LIN {X 0,Y 342.196,Z 1212.787,A -85,B 0,C 180,E1 21187.644,E2 21187.644} C_VEL
LIN {X 0,Y 370.541,Z 1183.05,A -85,B 0,C 180,E1 21194.239,E2 21194.239} C_VEL
LIN {X 0,Y 337.075,Z 1218.846,A -85,B 0,C 180,E1 21204.188,E2 21204.188} C_VEL
LIN {X 0,Y 317.104,Z 1240.275,A -85,B 0,C 180,E1 21216.022,E2 21216.022} C_VEL
LIN {X 0,Y 309.368,Z 1248.117,A -85,B 0,C 180,E1 21227.294,E2 21227.294} C_VEL
LIN {X 0,Y 299.7,Z 1248.319,A -85,B 0,C 180,E1 21233.729,E2 21233.729} C_VEL
LIN {X 0,Y 299.965,Z 1240.133,A -85,B 0,C 180,E1 21244.381,E2 21244.381} C_VEL
LIN {X 0,Y 304.172,Z 1219.099,A -85,B 0,C 180,E1 21255.958,E2 21255.958} C_VEL
LIN {X 0,Y 314.8,Z 1183.171,A -85,B 0,C 180,E1 21267.012,E2 21267.012} C_VEL
LIN {X 0,Y 330.638,Z 1134.667,A -85,B 0,C 180,E1 21275.905,E2 21275.905} C_VEL
LIN {X 0,Y 345.711,Z 1077.076,A -85,B 0,C 180,E1 21282.387,E2 21282.387} C_VEL
LIN {X 0,Y 328.382,Z 1020.895,A -85,B 0,C 180,E1 21289.392,E2 21289.392} C_VEL
LIN {X 0,Y 317.3,Z 992.068,A -85,B 0,C 180,E1 21293.134,E2 21293.134} C_VEL
LIN {X 0,Y 333.633,Z 1036.761,A -85,B 0,C 180,E1 21296.365,E2 21296.365} C_VEL
LIN {X 0,Y 329.633,Z 1087.019,A -85,B 0,C 180,E1 21298.729,E2 21298.729} C_VEL
LIN {X 0,Y 321.057,Z 1131.238,A -85,B 0,C 180,E1 21303.54,E2 21303.54} C_VEL
LIN {X 0,Y 311.784,Z 1164.217,A -85,B 0,C 180,E1 21310.381,E2 21310.381} C_VEL
LIN {X 0,Y 304.757,Z 1185.316,A -85,B 0,C 180,E1 21319.168,E2 21319.168} C_VEL
LIN {X 0,Y 302.413,Z 1192.13,A -85,B 0,C 180,E1 21328.492,E2 21328.492} C_VEL
LIN {X 0,Y 304.538,Z 1184.356,A -85,B 0,C 180,E1 21338.525,E2 21338.525} C_VEL
LIN {X 0,Y 311.172,Z 1162.189,A -85,B 0,C 180,E1 21347.305,E2 21347.305} C_VEL
LIN {X 0,Y 320.195,Z 1127.219,A -85,B 0,C 180,E1 21354.236,E2 21354.236} C_VEL
LIN {X 0,Y 327.949,Z 1082.319,A -85,B 0,C 180,E1 21358.849,E2 21358.849} C_VEL
LIN {X 0,Y 330.843,Z 1031.167,A -85,B 0,C 180,E1 21361.083,E2 21361.083} C_VEL
LIN {X 0,Y 306.991,Z 970.809,A -85,B 0,C 180,E1 21365.672,E2 21365.672} C_VEL
LIN {X 0,Y 296.216,Z 948.94,A -85,B 0,C 180,E1 21368,E2 21368} C_VEL
LIN {X 0,Y 296.219,Z 948.94,A -85,B 0,C 180,E1 21380.134,E2 21380.134} C_VEL
LIN {X 0,Y 296.775,Z 948.94,A -85,B 0,C 180,E1 21393.307,E2 21393.307} C_VEL
LIN {X 0,Y 298.047,Z 948.94,A -85,B 0,C 180,E1 21406.723,E2 21406.723} C_VEL
LIN {X 0,Y 298.821,Z 948.94,A -85,B 0,C 180,E1 21418.516,E2 21418.516} C_VEL
LIN {X 0,Y 297.907,Z 948.94,A -85,B 0,C 180,E1 21430.243,E2 21430.243} C_VEL
LIN {X 0,Y 297.236,Z 950.399,A -85,B 0,C 180,E1 21441.304,E2 21441.304} C_VEL
LIN {X 0,Y 327.096,Z 1016.083,A -85,B 0,C 180,E1 21452.614,E2 21452.614} C_VEL
LIN {X 0,Y 351.234,Z 1081.655,A -85,B 0,C 180,E1 21462.15,E2 21462.15} C_VEL
LIN {X 0,Y 328.608,Z 1154.976,A -85,B 0,C 180,E1 21469.978,E2 21469.978} C_VEL
LIN {X 0,Y 311.576,Z 1211.957,A -85,B 0,C 180,E1 21479.926,E2 21479.926} C_VEL
LIN {X 0,Y 302.573,Z 1251.413,A -85,B 0,C 180,E1 21491.052,E2 21491.052} C_VEL
LIN {X 0,Y 300.193,Z 1272.803,A -85,B 0,C 180,E1 21501.423,E2 21501.423} C_VEL
LIN {X 0,Y 299.986,Z 1281.152,A -85,B 0,C 180,E1 21511.521,E2 21511.521} C_VEL
LIN {X 0,Y 300.221,Z 1277.634,A -85,B 0,C 180,E1 21521.736,E2 21521.736} C_VEL
LIN {X 0,Y 307.735,Z 1258.286,A -85,B 0,C 180,E1 21534.221,E2 21534.221} C_VEL
LIN {X 0,Y 339.314,Z 1212.711,A -85,B 0,C 180,E1 21549.251,E2 21549.251} C_VEL
LIN {X 0,Y 361.602,Z 1191.419,A -85,B 0,C 180,E1 21554.373,E2 21554.373} C_VEL
LIN {X 0,Y 327.946,Z 1224.179,A -85,B 0,C 180,E1 21564.685,E2 21564.685} C_VEL
LIN {X 0,Y 307.047,Z 1244.419,A -85,B 0,C 180,E1 21578.268,E2 21578.268} C_VEL
LIN {X 0,Y 300.37,Z 1249.085,A -85,B 0,C 180,E1 21590.489,E2 21590.489} C_VEL
LIN {X 0,Y 299.7,Z 1248.319,A -85,B 0,C 180,E1 21593.729,E2 21593.729} C_VEL
LIN {X 0,Y 291.795,Z 1244.564,A -85,B 0,C 180,E1 21600.397,E2 21600.397} C_VEL
LIN {X 0,Y 294.315,Z 1227.603,A -85,B 0,C 180,E1 21612.345,E2 21612.345} C_VEL
LIN {X 0,Y 303.211,Z 1196.172,A -85,B 0,C 180,E1 21624.03,E2 21624.03} C_VEL
LIN {X 0,Y 317.833,Z 1152.021,A -85,B 0,C 180,E1 21633.753,E2 21633.753} C_VEL
LIN {X 0,Y 334.741,Z 1096.51,A -85,B 0,C 180,E1 21641.141,E2 21641.141} C_VEL
LIN {X 0,Y 337.819,Z 1076.712,A -85,B 0,C 180,E1 21643.202,E2 21643.202} C_VEL
LIN {X 0,Y 320.249,Z 1020.145,A -85,B 0,C 180,E1 21650.453,E2 21650.453} C_VEL
LIN {X 0,Y 313.932,Z 1002.402,A -85,B 0,C 180,E1 21652.96,E2 21652.96} C_VEL
LIN {X 0,Y 326.976,Z 1038.863,A -85,B 0,C 180,E1 21655.637,E2 21655.637} C_VEL
LIN {X 0,Y 322.812,Z 1088.072,A -85,B 0,C 180,E1 21658.019,E2 21658.019} C_VEL
LIN {X 0,Y 313.933,Z 1132.251,A -85,B 0,C 180,E1 21662.919,E2 21662.919} C_VEL
LIN {X 0,Y 303.873,Z 1166.286,A -85,B 0,C 180,E1 21670.229,E2 21670.229} C_VEL
LIN {X 0,Y 296.971,Z 1186.242,A -85,B 0,C 180,E1 21678.881,E2 21678.881} C_VEL
LIN {X 0,Y 294.475,Z 1193.081,A -85,B 0,C 180,E1 21688.451,E2 21688.451} C_VEL
LIN {X 0,Y 296.71,Z 1185.329,A -85,B 0,C 180,E1 21698.751,E2 21698.751} C_VEL
LIN {X 0,Y 303.512,Z 1163.552,A -85,B 0,C 180,E1 21707.65,E2 21707.65} C_VEL
LIN {X 0,Y 312.647,Z 1129.383,A -85,B 0,C 180,E1 21714.669,E2 21714.669} C_VEL
LIN {X 0,Y 320.8,Z 1085.261,A -85,B 0,C 180,E1 21719.404,E2 21719.404} C_VEL
LIN {X 0,Y 324.209,Z 1033.506,A -85,B 0,C 180,E1 21721.77,E2 21721.77} C_VEL
LIN {X 0,Y 300.618,Z 973.534,A -85,B 0,C 180,E1 21726.512,E2 21726.512} C_VEL
LIN {X 0,Y 288.132,Z 948.94,A -85,B 0,C 180,E1 21729.426,E2 21729.426} C_VEL
LIN {X 0,Y 288.256,Z 948.94,A -85,B 0,C 180,E1 21742.696,E2 21742.696} C_VEL
LIN {X 0,Y 288.788,Z 948.94,A -85,B 0,C 180,E1 21753.432,E2 21753.432} C_VEL
LIN {X 0,Y 289.956,Z 948.94,A -85,B 0,C 180,E1 21766.345,E2 21766.345} C_VEL
LIN {X 0,Y 290.838,Z 948.94,A -85,B 0,C 180,E1 21778.475,E2 21778.475} C_VEL
LIN {X 0,Y 289.84,Z 948.94,A -85,B 0,C 180,E1 21790.531,E2 21790.531} C_VEL
LIN {X 0,Y 289.433,Z 950.977,A -85,B 0,C 180,E1 21799.772,E2 21799.772} C_VEL
LIN {X 0,Y 318.268,Z 1014.18,A -85,B 0,C 180,E1 21811.209,E2 21811.209} C_VEL
LIN {X 0,Y 343.351,Z 1082.536,A -85,B 0,C 180,E1 21821.496,E2 21821.496} C_VEL
LIN {X 0,Y 320.993,Z 1155.423,A -85,B 0,C 180,E1 21829.546,E2 21829.546} C_VEL
LIN {X 0,Y 303.671,Z 1211.944,A -85,B 0,C 180,E1 21839.692,E2 21839.692} C_VEL
LIN {X 0,Y 294.557,Z 1251.213,A -85,B 0,C 180,E1 21851.101,E2 21851.101} C_VEL
LIN {X 0,Y 292.141,Z 1273.544,A -85,B 0,C 180,E1 21862.614,E2 21862.614} C_VEL
LIN {X 0,Y 292.001,Z 1280.42,A -85,B 0,C 180,E1 21871.562,E2 21871.562} C_VEL
LIN {X 0,Y 292.314,Z 1277.354,A -85,B 0,C 180,E1 21882.058,E2 21882.058} C_VEL
LIN {X 0,Y 301.034,Z 1257.777,A -85,B 0,C 180,E1 21895.446,E2 21895.446} C_VEL
LIN {X 0,Y 337.978,Z 1211.874,A -85,B 0,C 180,E1 21911.122,E2 21911.122} C_VEL
LIN {X 0,Y 352.937,Z 1198.914,A -85,B 0,C 180,E1 21914.182,E2 21914.182} C_VEL
LIN {X 0,Y 316.008,Z 1231.474,A -85,B 0,C 180,E1 21926.504,E2 21926.504} C_VEL
LIN {X 0,Y 297.02,Z 1247.559,A -85,B 0,C 180,E1 21940.631,E2 21940.631} C_VEL
LIN {X 0,Y 291.722,Z 1248.78,A -85,B 0,C 180,E1 21953.691,E2 21953.691} C_VEL
LIN {X 0,Y 291.795,Z 1244.564,A -85,B 0,C 180,E1 21960.397,E2 21960.397} C_VEL
LIN {X 0,Y 284.739,Z 1236.825,A -85,B 0,C 180,E1 21967.153,E2 21967.153} C_VEL
LIN {X 0,Y 290.083,Z 1212.471,A -85,B 0,C 180,E1 21979.119,E2 21979.119} C_VEL
LIN {X 0,Y 302.781,Z 1173.653,A -85,B 0,C 180,E1 21990.118,E2 21990.118} C_VEL
LIN {X 0,Y 320.044,Z 1122.033,A -85,B 0,C 180,E1 21998.853,E2 21998.853} C_VEL
LIN {X 0,Y 330.785,Z 1079.888,A -85,B 0,C 180,E1 22003.558,E2 22003.558} C_VEL
LIN {X 0,Y 313.837,Z 1023.996,A -85,B 0,C 180,E1 22010.973,E2 22010.973} C_VEL
LIN {X 0,Y 310.27,Z 1012.617,A -85,B 0,C 180,E1 22012.738,E2 22012.738} C_VEL
LIN {X 0,Y 320.333,Z 1041.652,A -85,B 0,C 180,E1 22014.893,E2 22014.893} C_VEL
LIN {X 0,Y 315.625,Z 1091.457,A -85,B 0,C 180,E1 22017.46,E2 22017.46} C_VEL
LIN {X 0,Y 306.576,Z 1134.252,A -85,B 0,C 180,E1 22022.42,E2 22022.42} C_VEL
LIN {X 0,Y 296.413,Z 1167.185,A -85,B 0,C 180,E1 22029.71,E2 22029.71} C_VEL
LIN {X 0,Y 289.181,Z 1187.17,A -85,B 0,C 180,E1 22038.577,E2 22038.577} C_VEL
LIN {X 0,Y 286.556,Z 1194.03,A -85,B 0,C 180,E1 22048.408,E2 22048.408} C_VEL
LIN {X 0,Y 288.861,Z 1186.306,A -85,B 0,C 180,E1 22058.991,E2 22058.991} C_VEL
LIN {X 0,Y 296.181,Z 1163.803,A -85,B 0,C 180,E1 22068.329,E2 22068.329} C_VEL
LIN {X 0,Y 305.803,Z 1129.297,A -85,B 0,C 180,E1 22075.456,E2 22075.456} C_VEL
LIN {X 0,Y 314.225,Z 1084.222,A -85,B 0,C 180,E1 22080.267,E2 22080.267} C_VEL
LIN {X 0,Y 316.797,Z 1033.119,A -85,B 0,C 180,E1 22082.658,E2 22082.658} C_VEL
LIN {X 0,Y 293.924,Z 975.892,A -85,B 0,C 180,E1 22087.46,E2 22087.46} C_VEL
LIN {X 0,Y 280.112,Z 948.94,A -85,B 0,C 180,E1 22090.95,E2 22090.95} C_VEL
LIN {X 0,Y 280.293,Z 948.94,A -85,B 0,C 180,E1 22105.312,E2 22105.312} C_VEL
LIN {X 0,Y 280.899,Z 948.94,A -85,B 0,C 180,E1 22116.06,E2 22116.06} C_VEL
LIN {X 0,Y 282.11,Z 948.94,A -85,B 0,C 180,E1 22129.115,E2 22129.115} C_VEL
LIN {X 0,Y 282.659,Z 948.94,A -85,B 0,C 180,E1 22141.508,E2 22141.508} C_VEL
LIN {X 0,Y 281.508,Z 948.94,A -85,B 0,C 180,E1 22154.01,E2 22154.01} C_VEL
LIN {X 0,Y 281.347,Z 950.523,A -85,B 0,C 180,E1 22157.992,E2 22157.992} C_VEL
LIN {X 0,Y 310.074,Z 1013.728,A -85,B 0,C 180,E1 22169.983,E2 22169.983} C_VEL
LIN {X 0,Y 334.573,Z 1080.888,A -85,B 0,C 180,E1 22180.455,E2 22180.455} C_VEL
LIN {X 0,Y 334.131,Z 1092.54,A -85,B 0,C 180,E1 22181.816,E2 22181.816} C_VEL
LIN {X 0,Y 310.895,Z 1163.485,A -85,B 0,C 180,E1 22190.258,E2 22190.258} C_VEL
LIN {X 0,Y 293.881,Z 1218.737,A -85,B 0,C 180,E1 22201.116,E2 22201.116} C_VEL
LIN {X 0,Y 285.978,Z 1255.72,A -85,B 0,C 180,E1 22213.112,E2 22213.112} C_VEL
LIN {X 0,Y 284.109,Z 1274.249,A -85,B 0,C 180,E1 22223.945,E2 22223.945} C_VEL
LIN {X 0,Y 283.672,Z 1280.07,A -85,B 0,C 180,E1 22234.678,E2 22234.678} C_VEL
LIN {X 0,Y 285.91,Z 1272.693,A -85,B 0,C 180,E1 22247.049,E2 22247.049} C_VEL
LIN {X 0,Y 302.716,Z 1245.944,A -85,B 0,C 180,E1 22261.838,E2 22261.838} C_VEL
LIN {X 0,Y 343.886,Z 1206.254,A -85,B 0,C 180,E1 22274.536,E2 22274.536} C_VEL
LIN {X 0,Y 307.499,Z 1235.138,A -85,B 0,C 180,E1 22286.657,E2 22286.657} C_VEL
LIN {X 0,Y 289.451,Z 1248.6,A -85,B 0,C 180,E1 22300.103,E2 22300.103} C_VEL
LIN {X 0,Y 283.988,Z 1249.777,A -85,B 0,C 180,E1 22312.352,E2 22312.352} C_VEL
LIN {X 0,Y 284.028,Z 1240.244,A -85,B 0,C 180,E1 22324.628,E2 22324.628} C_VEL
LIN {X 0,Y 284.739,Z 1236.825,A -85,B 0,C 180,E1 22327.153,E2 22327.153} C_VEL
LIN {X 0,Y 279.071,Z 1225.354,A -85,B 0,C 180,E1 22333.898,E2 22333.898} C_VEL
LIN {X 0,Y 289.115,Z 1191.74,A -85,B 0,C 180,E1 22346.116,E2 22346.116} C_VEL
LIN {X 0,Y 305.633,Z 1144.511,A -85,B 0,C 180,E1 22356.172,E2 22356.172} C_VEL
LIN {X 0,Y 323.653,Z 1086.172,A -85,B 0,C 180,E1 22363.538,E2 22363.538} C_VEL
LIN {X 0,Y 310.199,Z 1035.79,A -85,B 0,C 180,E1 22370.437,E2 22370.437} C_VEL
LIN {X 0,Y 306.497,Z 1022.683,A -85,B 0,C 180,E1 22372.489,E2 22372.489} C_VEL
LIN {X 0,Y 313.752,Z 1044.285,A -85,B 0,C 180,E1 22374.122,E2 22374.122} C_VEL
LIN {X 0,Y 308.721,Z 1093.794,A -85,B 0,C 180,E1 22376.8,E2 22376.8} C_VEL
LIN {X 0,Y 299.044,Z 1136.855,A -85,B 0,C 180,E1 22382.011,E2 22382.011} C_VEL
LIN {X 0,Y 288.492,Z 1169.258,A -85,B 0,C 180,E1 22389.529,E2 22389.529} C_VEL
LIN {X 0,Y 280.922,Z 1189.149,A -85,B 0,C 180,E1 22399.026,E2 22399.026} C_VEL
LIN {X 0,Y 278.645,Z 1194.978,A -85,B 0,C 180,E1 22408.363,E2 22408.363} C_VEL
LIN {X 0,Y 281.038,Z 1187.279,A -85,B 0,C 180,E1 22419.244,E2 22419.244} C_VEL
LIN {X 0,Y 288.65,Z 1164.809,A -85,B 0,C 180,E1 22428.825,E2 22428.825} C_VEL
LIN {X 0,Y 298.653,Z 1130.336,A -85,B 0,C 180,E1 22436.11,E2 22436.11} C_VEL
LIN {X 0,Y 307.275,Z 1086.268,A -85,B 0,C 180,E1 22440.945,E2 22440.945} C_VEL
LIN {X 0,Y 310.328,Z 1035.651,A -85,B 0,C 180,E1 22443.398,E2 22443.398} C_VEL
LIN {X 0,Y 287.811,Z 979.04,A -85,B 0,C 180,E1 22448.345,E2 22448.345} C_VEL
LIN {X 0,Y 271.994,Z 948.94,A -85,B 0,C 180,E1 22452.697,E2 22452.697} C_VEL
LIN {X 0,Y 272.115,Z 948.94,A -85,B 0,C 180,E1 22464.111,E2 22464.111} C_VEL
LIN {X 0,Y 272.911,Z 948.94,A -85,B 0,C 180,E1 22476.342,E2 22476.342} C_VEL
LIN {X 0,Y 274.047,Z 948.94,A -85,B 0,C 180,E1 22488.791,E2 22488.791} C_VEL
LIN {X 0,Y 274.647,Z 948.94,A -85,B 0,C 180,E1 22501.552,E2 22501.552} C_VEL
LIN {X 0,Y 273.423,Z 948.94,A -85,B 0,C 180,E1 22514.434,E2 22514.434} C_VEL
LIN {X 0,Y 273.525,Z 951.065,A -85,B 0,C 180,E1 22516.283,E2 22516.283} C_VEL
LIN {X 0,Y 299.882,Z 1008.76,A -85,B 0,C 180,E1 22527.884,E2 22527.884} C_VEL
LIN {X 0,Y 323.347,Z 1071.686,A -85,B 0,C 180,E1 22538.212,E2 22538.212} C_VEL
LIN {X 0,Y 327.574,Z 1091.222,A -85,B 0,C 180,E1 22541.025,E2 22541.025} C_VEL
LIN {X 0,Y 303.72,Z 1162.326,A -85,B 0,C 180,E1 22549.594,E2 22549.594} C_VEL
LIN {X 0,Y 286.233,Z 1217.541,A -85,B 0,C 180,E1 22560.633,E2 22560.633} C_VEL
LIN {X 0,Y 278.212,Z 1254.069,A -85,B 0,C 180,E1 22572.626,E2 22572.626} C_VEL
LIN {X 0,Y 276.165,Z 1273.149,A -85,B 0,C 180,E1 22583.77,E2 22583.77} C_VEL
LIN {X 0,Y 275.708,Z 1279.408,A -85,B 0,C 180,E1 22594.813,E2 22594.813} C_VEL
LIN {X 0,Y 278.122,Z 1272.742,A -85,B 0,C 180,E1 22607.541,E2 22607.541} C_VEL
LIN {X 0,Y 296.063,Z 1247.511,A -85,B 0,C 180,E1 22622.641,E2 22622.641} C_VEL
LIN {X 0,Y 335.06,Z 1212.825,A -85,B 0,C 180,E1 22634.409,E2 22634.409} C_VEL
LIN {X 0,Y 297.355,Z 1239.657,A -85,B 0,C 180,E1 22647.625,E2 22647.625} C_VEL
LIN {X 0,Y 279.662,Z 1250.736,A -85,B 0,C 180,E1 22662.664,E2 22662.664} C_VEL
LIN {X 0,Y 275.575,Z 1247.811,A -85,B 0,C 180,E1 22676.874,E2 22676.874} C_VEL
LIN {X 0,Y 277.111,Z 1234.507,A -85,B 0,C 180,E1 22688.852,E2 22688.852} C_VEL
LIN {X 0,Y 279.071,Z 1225.354,A -85,B 0,C 180,E1 22693.898,E2 22693.898} C_VEL
LIN {X 0,Y 275.012,Z 1210.369,A -85,B 0,C 180,E1 22700.518,E2 22700.518} C_VEL
LIN {X 0,Y 288.696,Z 1170.887,A -85,B 0,C 180,E1 22711.753,E2 22711.753} C_VEL
LIN {X 0,Y 307.411,Z 1117.161,A -85,B 0,C 180,E1 22720.802,E2 22720.802} C_VEL
LIN {X 0,Y 315.87,Z 1082.49,A -85,B 0,C 180,E1 22724.809,E2 22724.809} C_VEL
LIN {X 0,Y 302.185,Z 1032.745,A -85,B 0,C 180,E1 22732.153,E2 22732.153} C_VEL
LIN {X 0,Y 306.871,Z 1040.85,A -85,B 0,C 180,E1 22733.068,E2 22733.068} C_VEL
LIN {X 0,Y 302.676,Z 1091.179,A -85,B 0,C 180,E1 22735.695,E2 22735.695} C_VEL
LIN {X 0,Y 292.81,Z 1135.15,A -85,B 0,C 180,E1 22740.852,E2 22740.852} C_VEL
LIN {X 0,Y 281.548,Z 1168.987,A -85,B 0,C 180,E1 22748.587,E2 22748.587} C_VEL
LIN {X 0,Y 273.636,Z 1189.026,A -85,B 0,C 180,E1 22757.919,E2 22757.919} C_VEL
LIN {X 0,Y 270.725,Z 1195.927,A -85,B 0,C 180,E1 22768.315,E2 22768.315} C_VEL
LIN {X 0,Y 273.199,Z 1188.255,A -85,B 0,C 180,E1 22779.511,E2 22779.511} C_VEL
LIN {X 0,Y 281.13,Z 1165.864,A -85,B 0,C 180,E1 22789.332,E2 22789.332} C_VEL
LIN {X 0,Y 291.551,Z 1131.376,A -85,B 0,C 180,E1 22796.797,E2 22796.797} C_VEL
LIN {X 0,Y 300.491,Z 1087.432,A -85,B 0,C 180,E1 22801.72,E2 22801.72} C_VEL
LIN {X 0,Y 303.695,Z 1037.377,A -85,B 0,C 180,E1 22804.221,E2 22804.221} C_VEL
LIN {X 0,Y 281.389,Z 981.6,A -85,B 0,C 180,E1 22809.353,E2 22809.353} C_VEL
LIN {X 0,Y 263.874,Z 948.94,A -85,B 0,C 180,E1 22813.982,E2 22813.982} C_VEL
LIN {X 0,Y 264.171,Z 948.94,A -85,B 0,C 180,E1 22826.88,E2 22826.88} C_VEL
LIN {X 0,Y 265.129,Z 948.94,A -85,B 0,C 180,E1 22840.534,E2 22840.534} C_VEL
LIN {X 0,Y 266.207,Z 948.94,A -85,B 0,C 180,E1 22851.773,E2 22851.773} C_VEL
LIN {X 0,Y 266.634,Z 948.94,A -85,B 0,C 180,E1 22861.599,E2 22861.599} C_VEL
LIN {X 0,Y 265.695,Z 950.993,A -85,B 0,C 180,E1 22874.396,E2 22874.396} C_VEL
LIN {X 0,Y 291.171,Z 1006.99,A -85,B 0,C 180,E1 22886.268,E2 22886.268} C_VEL
LIN {X 0,Y 314.112,Z 1068.517,A -85,B 0,C 180,E1 22896.802,E2 22896.802} C_VEL
LIN {X 0,Y 320.316,Z 1092.024,A -85,B 0,C 180,E1 22900.415,E2 22900.415} C_VEL
LIN {X 0,Y 295.811,Z 1163.291,A -85,B 0,C 180,E1 22909.254,E2 22909.254} C_VEL
LIN {X 0,Y 278.213,Z 1217.712,A -85,B 0,C 180,E1 22920.504,E2 22920.504} C_VEL
LIN {X 0,Y 270.059,Z 1254.298,A -85,B 0,C 180,E1 22932.996,E2 22932.996} C_VEL
LIN {X 0,Y 268.223,Z 1271.947,A -85,B 0,C 180,E1 22943.584,E2 22943.584} C_VEL
LIN {X 0,Y 268.09,Z 1278.041,A -85,B 0,C 180,E1 22951.702,E2 22951.702} C_VEL
LIN {X 0,Y 269.043,Z 1275.444,A -85,B 0,C 180,E1 22964.784,E2 22964.784} C_VEL
LIN {X 0,Y 283.833,Z 1254.85,A -85,B 0,C 180,E1 22980.608,E2 22980.608} C_VEL
LIN {X 0,Y 325.181,Z 1219.676,A -85,B 0,C 180,E1 22994.376,E2 22994.376} C_VEL
LIN {X 0,Y 285.452,Z 1244.669,A -85,B 0,C 180,E1 23009.694,E2 23009.694} C_VEL
LIN {X 0,Y 270.197,Z 1251.943,A -85,B 0,C 180,E1 23025.39,E2 23025.39} C_VEL
LIN {X 0,Y 267.838,Z 1245.515,A -85,B 0,C 180,E1 23040.032,E2 23040.032} C_VEL
LIN {X 0,Y 270.573,Z 1227.527,A -85,B 0,C 180,E1 23052.999,E2 23052.999} C_VEL
LIN {X 0,Y 275.012,Z 1210.369,A -85,B 0,C 180,E1 23060.518,E2 23060.518} C_VEL
LIN {X 0,Y 273.629,Z 1192.009,A -85,B 0,C 180,E1 23066.893,E2 23066.893} C_VEL
LIN {X 0,Y 290.935,Z 1144.756,A -85,B 0,C 180,E1 23077.366,E2 23077.366} C_VEL
LIN {X 0,Y 309.095,Z 1086.931,A -85,B 0,C 180,E1 23084.982,E2 23084.982} C_VEL
LIN {X 0,Y 297.844,Z 1042.932,A -85,B 0,C 180,E1 23091.806,E2 23091.806} C_VEL
LIN {X 0,Y 300.904,Z 1046.549,A -85,B 0,C 180,E1 23092.391,E2 23092.391} C_VEL
LIN {X 0,Y 295.523,Z 1095.428,A -85,B 0,C 180,E1 23095.122,E2 23095.122} C_VEL
LIN {X 0,Y 285.23,Z 1138.164,A -85,B 0,C 180,E1 23100.438,E2 23100.438} C_VEL
LIN {X 0,Y 273.647,Z 1171.06,A -85,B 0,C 180,E1 23108.365,E2 23108.365} C_VEL
LIN {X 0,Y 265.366,Z 1191.011,A -85,B 0,C 180,E1 23118.374,E2 23118.374} C_VEL
LIN {X 0,Y 262.8,Z 1196.876,A -85,B 0,C 180,E1 23128.264,E2 23128.264} C_VEL
LIN {X 0,Y 265.384,Z 1189.23,A -85,B 0,C 180,E1 23139.794,E2 23139.794} C_VEL
LIN {X 0,Y 273.378,Z 1167.825,A -85,B 0,C 180,E1 23149.585,E2 23149.585} C_VEL
LIN {X 0,Y 284.128,Z 1133.707,A -85,B 0,C 180,E1 23157.306,E2 23157.306} C_VEL
LIN {X 0,Y 293.606,Z 1089.725,A -85,B 0,C 180,E1 23162.445,E2 23162.445} C_VEL
LIN {X 0,Y 297.247,Z 1039.608,A -85,B 0,C 180,E1 23165.048,E2 23165.048} C_VEL
LIN {X 0,Y 275.468,Z 984.861,A -85,B 0,C 180,E1 23170.309,E2 23170.309} C_VEL
LIN {X 0,Y 255.845,Z 948.94,A -85,B 0,C 180,E1 23176.232,E2 23176.232} C_VEL
LIN {X 0,Y 256.222,Z 948.94,A -85,B 0,C 180,E1 23189.728,E2 23189.728} C_VEL
LIN {X 0,Y 257.198,Z 948.94,A -85,B 0,C 180,E1 23201.025,E2 23201.025} C_VEL
LIN {X 0,Y 258.519,Z 948.94,A -85,B 0,C 180,E1 23214.915,E2 23214.915} C_VEL
LIN {X 0,Y 258.435,Z 948.94,A -85,B 0,C 180,E1 23225.021,E2 23225.021} C_VEL
LIN {X 0,Y 257.719,Z 950.484,A -85,B 0,C 180,E1 23232.295,E2 23232.295} C_VEL
LIN {X 0,Y 283.241,Z 1007.101,A -85,B 0,C 180,E1 23244.928,E2 23244.928} C_VEL
LIN {X 0,Y 306.031,Z 1068.305,A -85,B 0,C 180,E1 23255.837,E2 23255.837} C_VEL
LIN {X 0,Y 312.764,Z 1093.811,A -85,B 0,C 180,E1 23259.882,E2 23259.882} C_VEL
LIN {X 0,Y 287.432,Z 1165.597,A -85,B 0,C 180,E1 23269.133,E2 23269.133} C_VEL
LIN {X 0,Y 270.065,Z 1218.4,A -85,B 0,C 180,E1 23280.525,E2 23280.525} C_VEL
LIN {X 0,Y 262.088,Z 1253.606,A -85,B 0,C 180,E1 23292.971,E2 23292.971} C_VEL
LIN {X 0,Y 260.262,Z 1272.525,A -85,B 0,C 180,E1 23305.066,E2 23305.066} C_VEL
LIN {X 0,Y 259.731,Z 1277.992,A -85,B 0,C 180,E1 23315.11,E2 23315.11} C_VEL
LIN {X 0,Y 262.624,Z 1272.686,A -85,B 0,C 180,E1 23328.613,E2 23328.613} C_VEL
LIN {X 0,Y 286.288,Z 1247.577,A -85,B 0,C 180,E1 23345.752,E2 23345.752} C_VEL
LIN {X 0,Y 316.394,Z 1225.241,A -85,B 0,C 180,E1 23354.582,E2 23354.582} C_VEL
LIN {X 0,Y 276.151,Z 1247.578,A -85,B 0,C 180,E1 23370.388,E2 23370.388} C_VEL
LIN {X 0,Y 262.409,Z 1252.634,A -85,B 0,C 180,E1 23384.947,E2 23384.947} C_VEL
LIN {X 0,Y 259.838,Z 1245.597,A -85,B 0,C 180,E1 23400.033,E2 23400.033} C_VEL
LIN {X 0,Y 262.732,Z 1227.161,A -85,B 0,C 180,E1 23413.394,E2 23413.394} C_VEL
LIN {X 0,Y 273.115,Z 1193.643,A -85,B 0,C 180,E1 23426.421,E2 23426.421} C_VEL
LIN {X 0,Y 273.629,Z 1192.009,A -85,B 0,C 180,E1 23426.893,E2 23426.893} C_VEL
LIN {X 0,Y 273.689,Z 1170.801,A -85,B 0,C 180,E1 23432.86,E2 23432.86} C_VEL
LIN {X 0,Y 292.991,Z 1117.732,A -85,B 0,C 180,E1 23442.123,E2 23442.123} C_VEL
LIN {X 0,Y 301.193,Z 1086.084,A -85,B 0,C 180,E1 23445.973,E2 23445.973} C_VEL
LIN {X 0,Y 293.32,Z 1052.624,A -85,B 0,C 180,E1 23451.465,E2 23451.465} C_VEL
LIN {X 0,Y 288.029,Z 1101.865,A -85,B 0,C 180,E1 23454.756,E2 23454.756} C_VEL
LIN {X 0,Y 277.001,Z 1143.112,A -85,B 0,C 180,E1 23460.375,E2 23460.375} C_VEL
LIN {X 0,Y 264.797,Z 1175.265,A -85,B 0,C 180,E1 23468.928,E2 23468.928} C_VEL
LIN {X 0,Y 256.723,Z 1193.754,A -85,B 0,C 180,E1 23479.702,E2 23479.702} C_VEL
LIN {X 0,Y 255.297,Z 1197.206,A -85,B 0,C 180,E1 23491.619,E2 23491.619} C_VEL
LIN {X 0,Y 258.895,Z 1186.456,A -85,B 0,C 180,E1 23502.611,E2 23502.611} C_VEL
LIN {X 0,Y 268.426,Z 1161.53,A -85,B 0,C 180,E1 23512.343,E2 23512.343} C_VEL
LIN {X 0,Y 280.148,Z 1123.974,A -85,B 0,C 180,E1 23519.687,E2 23519.687} C_VEL
LIN {X 0,Y 288.775,Z 1078.334,A -85,B 0,C 180,E1 23524.198,E2 23524.198} C_VEL
LIN {X 0,Y 289.927,Z 1038.791,A -85,B 0,C 180,E1 23526.146,E2 23526.146} C_VEL
LIN {X 0,Y 268.667,Z 986.405,A -85,B 0,C 180,E1 23531.556,E2 23531.556} C_VEL
LIN {X 0,Y 247.787,Z 948.94,A -85,B 0,C 180,E1 23538.002,E2 23538.002} C_VEL
LIN {X 0,Y 248.297,Z 948.94,A -85,B 0,C 180,E1 23552.195,E2 23552.195} C_VEL
LIN {X 0,Y 249.467,Z 948.94,A -85,B 0,C 180,E1 23564.075,E2 23564.075} C_VEL
LIN {X 0,Y 250.775,Z 948.94,A -85,B 0,C 180,E1 23578.232,E2 23578.232} C_VEL
LIN {X 0,Y 249.913,Z 950.857,A -85,B 0,C 180,E1 23590.242,E2 23590.242} C_VEL
LIN {X 0,Y 273.802,Z 1003.728,A -85,B 0,C 180,E1 23602.799,E2 23602.799} C_VEL
LIN {X 0,Y 295.755,Z 1061.78,A -85,B 0,C 180,E1 23613.725,E2 23613.725} C_VEL
LIN {X 0,Y 304.954,Z 1096.211,A -85,B 0,C 180,E1 23619.413,E2 23619.413} C_VEL
LIN {X 0,Y 279.299,Z 1167.025,A -85,B 0,C 180,E1 23628.871,E2 23628.871} C_VEL
LIN {X 0,Y 261.495,Z 1220.663,A -85,B 0,C 180,E1 23641.02,E2 23641.02} C_VEL
LIN {X 0,Y 253.631,Z 1255.964,A -85,B 0,C 180,E1 23654.471,E2 23654.471} C_VEL
LIN {X 0,Y 252.272,Z 1272.942,A -85,B 0,C 180,E1 23666.637,E2 23666.637} C_VEL
LIN {X 0,Y 251.678,Z 1277.301,A -85,B 0,C 180,E1 23676.022,E2 23676.022} C_VEL
LIN {X 0,Y 256.106,Z 1271.187,A -85,B 0,C 180,E1 23690.911,E2 23690.911} C_VEL
LIN {X 0,Y 283.631,Z 1246.441,A -85,B 0,C 180,E1 23708.061,E2 23708.061} C_VEL
LIN {X 0,Y 306.388,Z 1231.114,A -85,B 0,C 180,E1 23714.539,E2 23714.539} C_VEL
LIN {X 0,Y 266.873,Z 1250.14,A -85,B 0,C 180,E1 23731.127,E2 23731.127} C_VEL
LIN {X 0,Y 253.128,Z 1252.732,A -85,B 0,C 180,E1 23747.92,E2 23747.92} C_VEL
LIN {X 0,Y 251.868,Z 1244.024,A -85,B 0,C 180,E1 23761.76,E2 23761.76} C_VEL
LIN {X 0,Y 255.774,Z 1223.281,A -85,B 0,C 180,E1 23775.523,E2 23775.523} C_VEL
LIN {X 0,Y 267.734,Z 1186.781,A -85,B 0,C 180,E1 23788.844,E2 23788.844} C_VEL
LIN {X 0,Y 273.689,Z 1170.801,A -85,B 0,C 180,E1 23792.86,E2 23792.86} C_VEL
LIN {X 0,Y 275.575,Z 1146.742,A -85,B 0,C 180,E1 23798.311,E2 23798.311} C_VEL
LIN {X 0,Y 294.167,Z 1089.524,A -85,B 0,C 180,E1 23806.3,E2 23806.3} C_VEL
LIN {X 0,Y 287.44,Z 1062.303,A -85,B 0,C 180,E1 23811.004,E2 23811.004} C_VEL
LIN {X 0,Y 279.997,Z 1109.974,A -85,B 0,C 180,E1 23814.588,E2 23814.588} C_VEL
LIN {X 0,Y 268.102,Z 1149.668,A -85,B 0,C 180,E1 23820.692,E2 23820.692} C_VEL
LIN {X 0,Y 256.461,Z 1178.264,A -85,B 0,C 180,E1 23829.119,E2 23829.119} C_VEL
LIN {X 0,Y 248.918,Z 1194.69,A -85,B 0,C 180,E1 23839.376,E2 23839.376} C_VEL
LIN {X 0,Y 247.369,Z 1198.163,A -85,B 0,C 180,E1 23851.671,E2 23851.671} C_VEL
LIN {X 0,Y 251.149,Z 1187.439,A -85,B 0,C 180,E1 23863.006,E2 23863.006} C_VEL
LIN {X 0,Y 261.1,Z 1162.538,A -85,B 0,C 180,E1 23873.005,E2 23873.005} C_VEL
LIN {X 0,Y 273.135,Z 1125.693,A -85,B 0,C 180,E1 23880.415,E2 23880.415} C_VEL
LIN {X 0,Y 282.257,Z 1079.483,A -85,B 0,C 180,E1 23885.102,E2 23885.102} C_VEL
LIN {X 0,Y 283.49,Z 1040.57,A -85,B 0,C 180,E1 23887.094,E2 23887.094} C_VEL
LIN {X 0,Y 262.594,Z 989.22,A -85,B 0,C 180,E1 23892.694,E2 23892.694} C_VEL
LIN {X 0,Y 239.717,Z 948.94,A -85,B 0,C 180,E1 23900.325,E2 23900.325} C_VEL
LIN {X 0,Y 240.229,Z 948.94,A -85,B 0,C 180,E1 23911.674,E2 23911.674} C_VEL
LIN {X 0,Y 241.584,Z 948.94,A -85,B 0,C 180,E1 23926.391,E2 23926.391} C_VEL
LIN {X 0,Y 242.764,Z 948.94,A -85,B 0,C 180,E1 23938.173,E2 23938.173} C_VEL
LIN {X 0,Y 242.039,Z 950.057,A -85,B 0,C 180,E1 23947.849,E2 23947.849} C_VEL
LIN {X 0,Y 265.232,Z 1002.065,A -85,B 0,C 180,E1 23960.922,E2 23960.922} C_VEL
LIN {X 0,Y 287.442,Z 1060.831,A -85,B 0,C 180,E1 23972.508,E2 23972.508} C_VEL
LIN {X 0,Y 297.408,Z 1097.595,A -85,B 0,C 180,E1 23978.826,E2 23978.826} C_VEL
LIN {X 0,Y 271.107,Z 1168.524,A -85,B 0,C 180,E1 23988.631,E2 23988.631} C_VEL
LIN {X 0,Y 253.293,Z 1221.193,A -85,B 0,C 180,E1 24001.065,E2 24001.065} C_VEL
LIN {X 0,Y 245.566,Z 1255.864,A -85,B 0,C 180,E1 24014.867,E2 24014.867} C_VEL
LIN {X 0,Y 244.361,Z 1271.739,A -85,B 0,C 180,E1 24026.528,E2 24026.528} C_VEL
LIN {X 0,Y 243.804,Z 1276.397,A -85,B 0,C 180,E1 24035.445,E2 24035.445} C_VEL
LIN {X 0,Y 247.235,Z 1272.518,A -85,B 0,C 180,E1 24049.819,E2 24049.819} C_VEL
LIN {X 0,Y 273.707,Z 1250.76,A -85,B 0,C 180,E1 24067.672,E2 24067.672} C_VEL
LIN {X 0,Y 297.169,Z 1235.932,A -85,B 0,C 180,E1 24075.092,E2 24075.092} C_VEL
LIN {X 0,Y 259.904,Z 1251.543,A -85,B 0,C 180,E1 24090.276,E2 24090.276} C_VEL
LIN {X 0,Y 245.248,Z 1253.288,A -85,B 0,C 180,E1 24107.526,E2 24107.526} C_VEL
LIN {X 0,Y 243.884,Z 1243.941,A -85,B 0,C 180,E1 24121.818,E2 24121.818} C_VEL
LIN {X 0,Y 247.972,Z 1222.667,A -85,B 0,C 180,E1 24136.024,E2 24136.024} C_VEL
LIN {X 0,Y 260.168,Z 1186.355,A -85,B 0,C 180,E1 24149.429,E2 24149.429} C_VEL
LIN {X 0,Y 275.575,Z 1146.742,A -85,B 0,C 180,E1 24158.311,E2 24158.311} C_VEL
LIN {X 0,Y 277.845,Z 1120.404,A -85,B 0,C 180,E1 24163.228,E2 24163.228} C_VEL
LIN {X 0,Y 286.54,Z 1090.077,A -85,B 0,C 180,E1 24167.117,E2 24167.117} C_VEL
LIN {X 0,Y 280.472,Z 1071.481,A -85,B 0,C 180,E1 24170.425,E2 24170.425} C_VEL
LIN {X 0,Y 271.758,Z 1118.147,A -85,B 0,C 180,E1 24174.505,E2 24174.505} C_VEL
LIN {X 0,Y 258.573,Z 1157.482,A -85,B 0,C 180,E1 24181.461,E2 24181.461} C_VEL
LIN {X 0,Y 246.467,Z 1184.593,A -85,B 0,C 180,E1 24191.052,E2 24191.052} C_VEL
LIN {X 0,Y 240.373,Z 1197.099,A -85,B 0,C 180,E1 24200.83,E2 24200.83} C_VEL
LIN {X 0,Y 239.445,Z 1199.119,A -85,B 0,C 180,E1 24211.726,E2 24211.726} C_VEL
LIN {X 0,Y 243.431,Z 1188.421,A -85,B 0,C 180,E1 24223.426,E2 24223.426} C_VEL
LIN {X 0,Y 253.818,Z 1163.547,A -85,B 0,C 180,E1 24233.705,E2 24233.705} C_VEL
LIN {X 0,Y 266.339,Z 1126.747,A -85,B 0,C 180,E1 24241.277,E2 24241.277} C_VEL
LIN {X 0,Y 275.894,Z 1080.108,A -85,B 0,C 180,E1 24246.083,E2 24246.083} C_VEL
LIN {X 0,Y 277.136,Z 1042.332,A -85,B 0,C 180,E1 24248.086,E2 24248.086} C_VEL
LIN {X 0,Y 256.221,Z 991.165,A -85,B 0,C 180,E1 24254.012,E2 24254.012} C_VEL
LIN {X 0,Y 231.711,Z 948.94,A -85,B 0,C 180,E1 24263.222,E2 24263.222} C_VEL
LIN {X 0,Y 232.333,Z 948.94,A -85,B 0,C 180,E1 24274.832,E2 24274.832} C_VEL
LIN {X 0,Y 233.663,Z 948.94,A -85,B 0,C 180,E1 24286.821,E2 24286.821} C_VEL
LIN {X 0,Y 234.763,Z 948.94,A -85,B 0,C 180,E1 24298.111,E2 24298.111} C_VEL
LIN {X 0,Y 234.442,Z 950.395,A -85,B 0,C 180,E1 24305.536,E2 24305.536} C_VEL
LIN {X 0,Y 257.384,Z 1002.206,A -85,B 0,C 180,E1 24319.337,E2 24319.337} C_VEL
LIN {X 0,Y 279.483,Z 1060.859,A -85,B 0,C 180,E1 24331.42,E2 24331.42} C_VEL
LIN {X 0,Y 289.779,Z 1099.223,A -85,B 0,C 180,E1 24338.243,E2 24338.243} C_VEL
LIN {X 0,Y 263.214,Z 1169.189,A -85,B 0,C 180,E1 24348.234,E2 24348.234} C_VEL
LIN {X 0,Y 245.161,Z 1221.566,A -85,B 0,C 180,E1 24361.079,E2 24361.079} C_VEL
LIN {X 0,Y 237.52,Z 1255.729,A -85,B 0,C 180,E1 24375.289,E2 24375.289} C_VEL
LIN {X 0,Y 236.381,Z 1272.05,A -85,B 0,C 180,E1 24388.252,E2 24388.252} C_VEL
LIN {X 0,Y 235.864,Z 1275.909,A -85,B 0,C 180,E1 24399.347,E2 24399.347} C_VEL
LIN {X 0,Y 244.581,Z 1268.274,A -85,B 0,C 180,E1 24415.944,E2 24415.944} C_VEL
LIN {X 0,Y 283.247,Z 1243.091,A -85,B 0,C 180,E1 24433.63,E2 24433.63} C_VEL
LIN {X 0,Y 286.73,Z 1240.921,A -85,B 0,C 180,E1 24435.445,E2 24435.445} C_VEL
LIN {X 0,Y 248.425,Z 1254.157,A -85,B 0,C 180,E1 24452.766,E2 24452.766} C_VEL
LIN {X 0,Y 236.296,Z 1252.226,A -85,B 0,C 180,E1 24470.796,E2 24470.796} C_VEL
LIN {X 0,Y 236.236,Z 1239.62,A -85,B 0,C 180,E1 24485.567,E2 24485.567} C_VEL
LIN {X 0,Y 242.115,Z 1214.777,A -85,B 0,C 180,E1 24499.885,E2 24499.885} C_VEL
LIN {X 0,Y 256.503,Z 1175.942,A -85,B 0,C 180,E1 24512.72,E2 24512.72} C_VEL
LIN {X 0,Y 276.414,Z 1124.347,A -85,B 0,C 180,E1 24522.67,E2 24522.67} C_VEL
LIN {X 0,Y 277.845,Z 1120.404,A -85,B 0,C 180,E1 24523.228,E2 24523.228} C_VEL
LIN {X 0,Y 280.209,Z 1099.166,A -85,B 0,C 180,E1 24526.501,E2 24526.501} C_VEL
LIN {X 0,Y 279.225,Z 1092.201,A -85,B 0,C 180,E1 24527.685,E2 24527.685} C_VEL
LIN {X 0,Y 275.431,Z 1082.54,A -85,B 0,C 180,E1 24529.563,E2 24529.563} C_VEL
LIN {X 0,Y 272.37,Z 1085.422,A -85,B 0,C 180,E1 24530.189,E2 24530.189} C_VEL
LIN {X 0,Y 261.592,Z 1131.211,A -85,B 0,C 180,E1 24535.21,E2 24535.21} C_VEL
LIN {X 0,Y 247.947,Z 1167.156,A -85,B 0,C 180,E1 24543.076,E2 24543.076} C_VEL
LIN {X 0,Y 236.707,Z 1190.053,A -85,B 0,C 180,E1 24553.14,E2 24553.14} C_VEL
LIN {X 0,Y 231.51,Z 1199.995,A -85,B 0,C 180,E1 24564.265,E2 24564.265} C_VEL
LIN {X 0,Y 231.783,Z 1198.316,A -85,B 0,C 180,E1 24575.542,E2 24575.542} C_VEL
LIN {X 0,Y 238.444,Z 1183.403,A -85,B 0,C 180,E1 24587.284,E2 24587.284} C_VEL
LIN {X 0,Y 250.167,Z 1155.225,A -85,B 0,C 180,E1 24596.961,E2 24596.961} C_VEL
LIN {X 0,Y 262.94,Z 1115.309,A -85,B 0,C 180,E1 24603.889,E2 24603.889} C_VEL
LIN {X 0,Y 271.218,Z 1067.818,A -85,B 0,C 180,E1 24607.865,E2 24607.865} C_VEL
LIN {X 0,Y 270.587,Z 1043.344,A -85,B 0,C 180,E1 24609.2,E2 24609.2} C_VEL
LIN {X 0,Y 250.112,Z 993.656,A -85,B 0,C 180,E1 24615.343,E2 24615.343} C_VEL
LIN {X 0,Y 226.452,Z 955.004,A -85,B 0,C 180,E1 24624.195,E2 24624.195} C_VEL
LIN {X 0,Y 223.758,Z 948.94,A -85,B 0,C 180,E1 24626.35,E2 24626.35} C_VEL
LIN {X 0,Y 224.566,Z 948.94,A -85,B 0,C 180,E1 24638.136,E2 24638.136} C_VEL
LIN {X 0,Y 225.893,Z 948.94,A -85,B 0,C 180,E1 24650.291,E2 24650.291} C_VEL
LIN {X 0,Y 226.549,Z 950.215,A -85,B 0,C 180,E1 24662.843,E2 24662.843} C_VEL
LIN {X 0,Y 248.223,Z 998.924,A -85,B 0,C 180,E1 24676.849,E2 24676.849} C_VEL
LIN {X 0,Y 269.871,Z 1056.205,A -85,B 0,C 180,E1 24689.352,E2 24689.352} C_VEL
LIN {X 0,Y 282.558,Z 1099.761,A -85,B 0,C 180,E1 24697.53,E2 24697.53} C_VEL
LIN {X 0,Y 255.521,Z 1169.375,A -85,B 0,C 180,E1 24707.732,E2 24707.732} C_VEL
LIN {X 0,Y 237.325,Z 1220.888,A -85,B 0,C 180,E1 24720.768,E2 24720.768} C_VEL
LIN {X 0,Y 229.723,Z 1253.922,A -85,B 0,C 180,E1 24734.778,E2 24734.778} C_VEL
LIN {X 0,Y 228.542,Z 1269.25,A -85,B 0,C 180,E1 24746.308,E2 24746.308} C_VEL
LIN {X 0,Y 227.891,Z 1274.585,A -85,B 0,C 180,E1 24755.826,E2 24755.826} C_VEL
LIN {X 0,Y 233.455,Z 1271.153,A -85,B 0,C 180,E1 24773.051,E2 24773.051} C_VEL
LIN {X 0,Y 267.648,Z 1250.224,A -85,B 0,C 180,E1 24791.874,E2 24791.874} C_VEL
LIN {X 0,Y 278.098,Z 1244.735,A -85,B 0,C 180,E1 24795.278,E2 24795.278} C_VEL
LIN {X 0,Y 241.293,Z 1255.311,A -85,B 0,C 180,E1 24811.891,E2 24811.891} C_VEL
LIN {X 0,Y 228.346,Z 1252.485,A -85,B 0,C 180,E1 24830.472,E2 24830.472} C_VEL
LIN {X 0,Y 228.276,Z 1239.363,A -85,B 0,C 180,E1 24845.761,E2 24845.761} C_VEL
LIN {X 0,Y 234.702,Z 1213.128,A -85,B 0,C 180,E1 24860.874,E2 24860.874} C_VEL
LIN {X 0,Y 250.329,Z 1172.516,A -85,B 0,C 180,E1 24874.156,E2 24874.156} C_VEL
LIN {X 0,Y 271.072,Z 1119.487,A -85,B 0,C 180,E1 24884.122,E2 24884.122} C_VEL
LIN {X 0,Y 279.225,Z 1092.201,A -85,B 0,C 180,E1 24887.685,E2 24887.685} C_VEL
LIN {X 0,Y 272.702,Z 1093.488,A -85,B 0,C 180,E1 24889.372,E2 24889.372} C_VEL
LIN {X 0,Y 260.517,Z 1113.903,A -85,B 0,C 180,E1 24891.727,E2 24891.727} C_VEL
LIN {X 0,Y 246.84,Z 1154.085,A -85,B 0,C 180,E1 24898.4,E2 24898.4} C_VEL
LIN {X 0,Y 233.304,Z 1182.89,A -85,B 0,C 180,E1 24907.942,E2 24907.942} C_VEL
LIN {X 0,Y 224.708,Z 1198.977,A -85,B 0,C 180,E1 24920.185,E2 24920.185} C_VEL
LIN {X 0,Y 223.589,Z 1201.032,A -85,B 0,C 180,E1 24931.848,E2 24931.848} C_VEL
LIN {X 0,Y 228.085,Z 1190.319,A -85,B 0,C 180,E1 24944.39,E2 24944.39} C_VEL
LIN {X 0,Y 239.366,Z 1165.563,A -85,B 0,C 180,E1 24955.233,E2 24955.233} C_VEL
LIN {X 0,Y 252.91,Z 1128.98,A -85,B 0,C 180,E1 24963.12,E2 24963.12} C_VEL
LIN {X 0,Y 263.185,Z 1082.973,A -85,B 0,C 180,E1 24968.07,E2 24968.07} C_VEL
LIN {X 0,Y 264.832,Z 1046.606,A -85,B 0,C 180,E1 24970.157,E2 24970.157} C_VEL
LIN {X 0,Y 244.853,Z 997.438,A -85,B 0,C 180,E1 24976.501,E2 24976.501} C_VEL
LIN {X 0,Y 222.037,Z 960.169,A -85,B 0,C 180,E1 24985.589,E2 24985.589} C_VEL
LIN {X 0,Y 215.866,Z 948.94,A -85,B 0,C 180,E1 24989.789,E2 24989.789} C_VEL
LIN {X 0,Y 217.414,Z 948.94,A -85,B 0,C 180,E1 25005.817,E2 25005.817} C_VEL
LIN {X 0,Y 218.587,Z 949.499,A -85,B 0,C 180,E1 25019.762,E2 25019.762} C_VEL
LIN {X 0,Y 237.818,Z 992.498,A -85,B 0,C 180,E1 25033.34,E2 25033.34} C_VEL
LIN {X 0,Y 259.571,Z 1049.261,A -85,B 0,C 180,E1 25046.676,E2 25046.676} C_VEL
LIN {X 0,Y 274.79,Z 1101.688,A -85,B 0,C 180,E1 25056.94,E2 25056.94} C_VEL
LIN {X 0,Y 247.255,Z 1171.001,A -85,B 0,C 180,E1 25067.529,E2 25067.529} C_VEL
LIN {X 0,Y 228.759,Z 1222.862,A -85,B 0,C 180,E1 25081.365,E2 25081.365} C_VEL
LIN {X 0,Y 221.43,Z 1255.315,A -85,B 0,C 180,E1 25096.224,E2 25096.224} C_VEL
LIN {X 0,Y 220.569,Z 1269.501,A -85,B 0,C 180,E1 25108.126,E2 25108.126} C_VEL
LIN {X 0,Y 219.989,Z 1274.304,A -85,B 0,C 180,E1 25120.028,E2 25120.028} C_VEL
LIN {X 0,Y 232.216,Z 1267.294,A -85,B 0,C 180,E1 25139.449,E2 25139.449} C_VEL
LIN {X 0,Y 269.091,Z 1248.34,A -85,B 0,C 180,E1 25155.21,E2 25155.21} C_VEL
LIN {X 0,Y 229.879,Z 1256.702,A -85,B 0,C 180,E1 25174.626,E2 25174.626} C_VEL
LIN {X 0,Y 219.713,Z 1250.318,A -85,B 0,C 180,E1 25194.091,E2 25194.091} C_VEL
LIN {X 0,Y 221.094,Z 1235.064,A -85,B 0,C 180,E1 25208.925,E2 25208.925} C_VEL
LIN {X 0,Y 229.762,Z 1205.224,A -85,B 0,C 180,E1 25224.426,E2 25224.426} C_VEL
LIN {X 0,Y 248.158,Z 1159.948,A -85,B 0,C 180,E1 25237.679,E2 25237.679} C_VEL
LIN {X 0,Y 269.771,Z 1103.668,A -85,B 0,C 180,E1 25247.029,E2 25247.029} C_VEL
LIN {X 0,Y 271.506,Z 1091.972,A -85,B 0,C 180,E1 25248.681,E2 25248.681} C_VEL
LIN {X 0,Y 265.076,Z 1093.401,A -85,B 0,C 180,E1 25249.674,E2 25249.674} C_VEL
LIN {X 0,Y 260.517,Z 1113.903,A -85,B 0,C 180,E1 25251.727,E2 25251.727} C_VEL
LIN {X 0,Y 248.45,Z 1133.553,A -85,B 0,C 180,E1 25253.223,E2 25253.223} C_VEL
LIN {X 0,Y 234.079,Z 1168.471,A -85,B 0,C 180,E1 25261.163,E2 25261.163} C_VEL
LIN {X 0,Y 221.537,Z 1191.904,A -85,B 0,C 180,E1 25271.948,E2 25271.948} C_VEL
LIN {X 0,Y 215.731,Z 1201.881,A -85,B 0,C 180,E1 25283.844,E2 25283.844} C_VEL
LIN {X 0,Y 215.998,Z 1200.244,A -85,B 0,C 180,E1 25295.948,E2 25295.948} C_VEL
LIN {X 0,Y 223.59,Z 1184.958,A -85,B 0,C 180,E1 25308.703,E2 25308.703} C_VEL
LIN {X 0,Y 236.815,Z 1155.565,A -85,B 0,C 180,E1 25319.14,E2 25319.14} C_VEL
LIN {X 0,Y 250.385,Z 1115.821,A -85,B 0,C 180,E1 25326.109,E2 25326.109} C_VEL
LIN {X 0,Y 259.134,Z 1068.18,A -85,B 0,C 180,E1 25330.125,E2 25330.125} C_VEL
LIN {X 0,Y 258.309,Z 1046.976,A -85,B 0,C 180,E1 25331.436,E2 25331.436} C_VEL
LIN {X 0,Y 238.421,Z 998.788,A -85,B 0,C 180,E1 25338.175,E2 25338.175} C_VEL
LIN {X 0,Y 215.785,Z 961.969,A -85,B 0,C 180,E1 25348.114,E2 25348.114} C_VEL
LIN {X 0,Y 208.004,Z 948.94,A -85,B 0,C 180,E1 25353.641,E2 25353.641} C_VEL
LIN {X 0,Y 209.731,Z 948.94,A -85,B 0,C 180,E1 25369.535,E2 25369.535} C_VEL
LIN {X 0,Y 210.752,Z 951.03,A -85,B 0,C 180,E1 25376.863,E2 25376.863} C_VEL
LIN {X 0,Y 226.537,Z 984.246,A -85,B 0,C 180,E1 25388.838,E2 25388.838} C_VEL
LIN {X 0,Y 246.515,Z 1035.037,A -85,B 0,C 180,E1 25402.118,E2 25402.118} C_VEL
LIN {X 0,Y 265.231,Z 1092.594,A -85,B 0,C 180,E1 25414.33,E2 25414.33} C_VEL
LIN {X 0,Y 266.383,Z 1105.089,A -85,B 0,C 180,E1 25416.52,E2 25416.52} C_VEL
LIN {X 0,Y 239.087,Z 1172.295,A -85,B 0,C 180,E1 25427.253,E2 25427.253} C_VEL
LIN {X 0,Y 220.68,Z 1222.885,A -85,B 0,C 180,E1 25441.342,E2 25441.342} C_VEL
LIN {X 0,Y 213.399,Z 1255.036,A -85,B 0,C 180,E1 25456.743,E2 25456.743} C_VEL
LIN {X 0,Y 212.572,Z 1269.645,A -85,B 0,C 180,E1 25470.095,E2 25470.095} C_VEL
LIN {X 0,Y 213.372,Z 1273.357,A -85,B 0,C 180,E1 25486.339,E2 25486.339} C_VEL
LIN {X 0,Y 237.342,Z 1261.483,A -85,B 0,C 180,E1 25507.509,E2 25507.509} C_VEL
LIN {X 0,Y 259.171,Z 1251.801,A -85,B 0,C 180,E1 25515.407,E2 25515.407} C_VEL
LIN {X 0,Y 222.611,Z 1257.62,A -85,B 0,C 180,E1 25533.736,E2 25533.736} C_VEL
LIN {X 0,Y 211.73,Z 1250.343,A -85,B 0,C 180,E1 25553.868,E2 25553.868} C_VEL
LIN {X 0,Y 213.186,Z 1234.453,A -85,B 0,C 180,E1 25569.258,E2 25569.258} C_VEL
LIN {X 0,Y 222.415,Z 1203.863,A -85,B 0,C 180,E1 25585.289,E2 25585.289} C_VEL
LIN {X 0,Y 240.972,Z 1159.288,A -85,B 0,C 180,E1 25598.507,E2 25598.507} C_VEL
LIN {X 0,Y 263.732,Z 1101.128,A -85,B 0,C 180,E1 25608.188,E2 25608.188} C_VEL
LIN {X 0,Y 257.25,Z 1102.68,A -85,B 0,C 180,E1 25609.301,E2 25609.301} C_VEL
LIN {X 0,Y 248.45,Z 1133.553,A -85,B 0,C 180,E1 25613.223,E2 25613.223} C_VEL
LIN {X 0,Y 235.337,Z 1151.514,A -85,B 0,C 180,E1 25615.359,E2 25615.359} C_VEL
LIN {X 0,Y 219.783,Z 1182.807,A -85,B 0,C 180,E1 25625.423,E2 25625.423} C_VEL
LIN {X 0,Y 209.853,Z 1199.617,A -85,B 0,C 180,E1 25637.72,E2 25637.72} C_VEL
LIN {X 0,Y 207.725,Z 1202.947,A -85,B 0,C 180,E1 25651.99,E2 25651.99} C_VEL
LIN {X 0,Y 213.315,Z 1191.162,A -85,B 0,C 180,E1 25666.212,E2 25666.212} C_VEL
LIN {X 0,Y 225.766,Z 1166.169,A -85,B 0,C 180,E1 25677.412,E2 25677.412} C_VEL
LIN {X 0,Y 240.588,Z 1128.548,A -85,B 0,C 180,E1 25685.577,E2 25685.577} C_VEL
LIN {X 0,Y 251.405,Z 1082.164,A -85,B 0,C 180,E1 25690.531,E2 25690.531} C_VEL
LIN {X 0,Y 252.855,Z 1050.751,A -85,B 0,C 180,E1 25692.439,E2 25692.439} C_VEL
LIN {X 0,Y 233.768,Z 1003.522,A -85,B 0,C 180,E1 25699.303,E2 25699.303} C_VEL
LIN {X 0,Y 212.311,Z 967.966,A -85,B 0,C 180,E1 25709.332,E2 25709.332} C_VEL
LIN {X 0,Y 200.395,Z 948.94,A -85,B 0,C 180,E1 25718.869,E2 25718.869} C_VEL
LIN {X 0,Y 202.256,Z 950.794,A -85,B 0,C 180,E1 25732.953,E2 25732.953} C_VEL
LIN {X 0,Y 216.862,Z 979.079,A -85,B 0,C 180,E1 25744.844,E2 25744.844} C_VEL
LIN {X 0,Y 235.953,Z 1027.643,A -85,B 0,C 180,E1 25758.724,E2 25758.724} C_VEL
LIN {X 0,Y 254.173,Z 1082.309,A -85,B 0,C 180,E1 25771.119,E2 25771.119} C_VEL
LIN {X 0,Y 258.951,Z 1105.973,A -85,B 0,C 180,E1 25775.788,E2 25775.788} C_VEL
LIN {X 0,Y 230.717,Z 1174.169,A -85,B 0,C 180,E1 25787.104,E2 25787.104} C_VEL
LIN {X 0,Y 212.201,Z 1224.179,A -85,B 0,C 180,E1 25801.84,E2 25801.84} C_VEL
LIN {X 0,Y 205.389,Z 1254.702,A -85,B 0,C 180,E1 25817.303,E2 25817.303} C_VEL
LIN {X 0,Y 204.7,Z 1268.302,A -85,B 0,C 180,E1 25830.105,E2 25830.105} C_VEL
LIN {X 0,Y 204.993,Z 1272.779,A -85,B 0,C 180,E1 25845.122,E2 25845.122} C_VEL
LIN {X 0,Y 227.32,Z 1263.631,A -85,B 0,C 180,E1 25867.011,E2 25867.011} C_VEL
LIN {X 0,Y 249.272,Z 1254.818,A -85,B 0,C 180,E1 25875.602,E2 25875.602} C_VEL
LIN {X 0,Y 211.415,Z 1257.825,A -85,B 0,C 180,E1 25896.787,E2 25896.787} C_VEL
LIN {X 0,Y 203.633,Z 1248.701,A -85,B 0,C 180,E1 25915.767,E2 25915.767} C_VEL
LIN {X 0,Y 205.855,Z 1230.754,A -85,B 0,C 180,E1 25931.741,E2 25931.741} C_VEL
LIN {X 0,Y 216.969,Z 1198.084,A -85,B 0,C 180,E1 25947.875,E2 25947.875} C_VEL
LIN {X 0,Y 237.214,Z 1150.832,A -85,B 0,C 180,E1 25961.031,E2 25961.031} C_VEL
LIN {X 0,Y 252.951,Z 1108.999,A -85,B 0,C 180,E1 25968.181,E2 25968.181} C_VEL
LIN {X 0,Y 249.604,Z 1110.495,A -85,B 0,C 180,E1 25968.872,E2 25968.872} C_VEL
LIN {X 0,Y 235.337,Z 1151.514,A -85,B 0,C 180,E1 25975.359,E2 25975.359} C_VEL
LIN {X 0,Y 218.078,Z 1174.411,A -85,B 0,C 180,E1 25980.641,E2 25980.641} C_VEL
LIN {X 0,Y 204.933,Z 1196.289,A -85,B 0,C 180,E1 25992.664,E2 25992.664} C_VEL
LIN {X 0,Y 199.96,Z 1203.767,A -85,B 0,C 180,E1 26003.357,E2 26003.357} C_VEL
LIN {X 0,Y 200.226,Z 1202.171,A -85,B 0,C 180,E1 26016.419,E2 26016.419} C_VEL
LIN {X 0,Y 208.629,Z 1186.937,A -85,B 0,C 180,E1 26030.099,E2 26030.099} C_VEL
LIN {X 0,Y 223.173,Z 1157.488,A -85,B 0,C 180,E1 26041.149,E2 26041.149} C_VEL
LIN {X 0,Y 237.757,Z 1117.972,A -85,B 0,C 180,E1 26048.362,E2 26048.362} C_VEL
LIN {X 0,Y 247.322,Z 1069.807,A -85,B 0,C 180,E1 26052.537,E2 26052.537} C_VEL
LIN {X 0,Y 246.479,Z 1051.11,A -85,B 0,C 180,E1 26053.863,E2 26053.863} C_VEL
LIN {X 0,Y 227.587,Z 1004.951,A -85,B 0,C 180,E1 26061.167,E2 26061.167} C_VEL
LIN {X 0,Y 206.542,Z 969.934,A -85,B 0,C 180,E1 26072.167,E2 26072.167} C_VEL
LIN {X 0,Y 195.188,Z 954.699,A -85,B 0,C 180,E1 26081.702,E2 26081.702} C_VEL
LIN {X 0,Y 193.182,Z 948.94,A -85,B 0,C 180,E1 26086.213,E2 26086.213} C_VEL
LIN {X 0,Y 197.768,Z 956.922,A -85,B 0,C 180,E1 26092.238,E2 26092.238} C_VEL
LIN {X 0,Y 212.118,Z 985.813,A -85,B 0,C 180,E1 26104.577,E2 26104.577} C_VEL
LIN {X 0,Y 230.524,Z 1034.255,A -85,B 0,C 180,E1 26118.683,E2 26118.683} C_VEL
LIN {X 0,Y 247.988,Z 1088.547,A -85,B 0,C 180,E1 26131.308,E2 26131.308} C_VEL
LIN {X 0,Y 251.266,Z 1107.516,A -85,B 0,C 180,E1 26135.109,E2 26135.109} C_VEL
LIN {X 0,Y 222.528,Z 1175.281,A -85,B 0,C 180,E1 26146.811,E2 26146.811} C_VEL
LIN {X 0,Y 203.742,Z 1225.24,A -85,B 0,C 180,E1 26162.313,E2 26162.313} C_VEL
LIN {X 0,Y 197.315,Z 1255.806,A -85,B 0,C 180,E1 26179.027,E2 26179.027} C_VEL
LIN {X 0,Y 196.7,Z 1268.302,A -85,B 0,C 180,E1 26192.319,E2 26192.319} C_VEL
LIN {X 0,Y 199.032,Z 1271.653,A -85,B 0,C 180,E1 26210.177,E2 26210.177} C_VEL
LIN {X 0,Y 228.926,Z 1261.247,A -85,B 0,C 180,E1 26231.637,E2 26231.637} C_VEL
LIN {X 0,Y 239.257,Z 1257.431,A -85,B 0,C 180,E1 26235.797,E2 26235.797} C_VEL
LIN {X 0,Y 203.983,Z 1258.378,A -85,B 0,C 180,E1 26255.888,E2 26255.888} C_VEL
LIN {X 0,Y 195.672,Z 1248.466,A -85,B 0,C 180,E1 26275.595,E2 26275.595} C_VEL
LIN {X 0,Y 198.019,Z 1229.905,A -85,B 0,C 180,E1 26292.212,E2 26292.212} C_VEL
LIN {X 0,Y 210.433,Z 1194.968,A -85,B 0,C 180,E1 26309.464,E2 26309.464} C_VEL
LIN {X 0,Y 231.932,Z 1145.919,A -85,B 0,C 180,E1 26322.812,E2 26322.812} C_VEL
LIN {X 0,Y 242.748,Z 1116.301,A -85,B 0,C 180,E1 26328.107,E2 26328.107} C_VEL
LIN {X 0,Y 226.04,Z 1158.419,A -85,B 0,C 180,E1 26335.68,E2 26335.68} C_VEL
LIN {X 0,Y 218.078,Z 1174.411,A -85,B 0,C 180,E1 26340.641,E2 26340.641} C_VEL
LIN {X 0,Y 200.906,Z 1191.729,A -85,B 0,C 180,E1 26347.684,E2 26347.684} C_VEL
LIN {X 0,Y 193.156,Z 1203.168,A -85,B 0,C 180,E1 26359.423,E2 26359.423} C_VEL
LIN {X 0,Y 191.868,Z 1204.86,A -85,B 0,C 180,E1 26372.154,E2 26372.154} C_VEL
LIN {X 0,Y 197.468,Z 1194.308,A -85,B 0,C 180,E1 26386.633,E2 26386.633} C_VEL
LIN {X 0,Y 211.09,Z 1169.595,A -85,B 0,C 180,E1 26398.908,E2 26398.908} C_VEL
LIN {X 0,Y 226.964,Z 1133.338,A -85,B 0,C 180,E1 26407.471,E2 26407.471} C_VEL
LIN {X 0,Y 239.167,Z 1086.877,A -85,B 0,C 180,E1 26412.809,E2 26412.809} C_VEL
LIN {X 0,Y 241.316,Z 1055.268,A -85,B 0,C 180,E1 26414.911,E2 26414.911} C_VEL
LIN {X 0,Y 223.41,Z 1010.148,A -85,B 0,C 180,E1 26422.308,E2 26422.308} C_VEL
LIN {X 0,Y 203.738,Z 976.579,A -85,B 0,C 180,E1 26433.253,E2 26433.253} C_VEL
LIN {X 0,Y 192.63,Z 960.936,A -85,B 0,C 180,E1 26443.505,E2 26443.505} C_VEL
LIN {X 0,Y 190.067,Z 956.898,A -85,B 0,C 180,E1 26447.414,E2 26447.414} C_VEL
LIN {X 0,Y 203.536,Z 983.156,A -85,B 0,C 180,E1 26460.905,E2 26460.905} C_VEL
LIN {X 0,Y 220.848,Z 1028.616,A -85,B 0,C 180,E1 26475.405,E2 26475.405} C_VEL
LIN {X 0,Y 238.862,Z 1084.213,A -85,B 0,C 180,E1 26489.164,E2 26489.164} C_VEL
LIN {X 0,Y 244.233,Z 1107.648,A -85,B 0,C 180,E1 26494.232,E2 26494.232} C_VEL
LIN {X 0,Y 214.778,Z 1175.347,A -85,B 0,C 180,E1 26506.255,E2 26506.255} C_VEL
LIN {X 0,Y 195.474,Z 1225.583,A -85,B 0,C 180,E1 26522.554,E2 26522.554} C_VEL
LIN {X 0,Y 189.393,Z 1255.341,A -85,B 0,C 180,E1 26539.731,E2 26539.731} C_VEL
LIN {X 0,Y 188.812,Z 1266.884,A -85,B 0,C 180,E1 26552.416,E2 26552.416} C_VEL
LIN {X 0,Y 191.416,Z 1270.917,A -85,B 0,C 180,E1 26571.017,E2 26571.017} C_VEL
LIN {X 0,Y 227.529,Z 1260.386,A -85,B 0,C 180,E1 26594.574,E2 26594.574} C_VEL
LIN {X 0,Y 229.145,Z 1259.63,A -85,B 0,C 180,E1 26595.985,E2 26595.985} C_VEL
LIN {X 0,Y 193.087,Z 1257.472,A -85,B 0,C 180,E1 26619.331,E2 26619.331} C_VEL
LIN {X 0,Y 187.847,Z 1244.146,A -85,B 0,C 180,E1 26640.045,E2 26640.045} C_VEL
LIN {X 0,Y 192.537,Z 1220.748,A -85,B 0,C 180,E1 26657.89,E2 26657.89} C_VEL
LIN {X 0,Y 207.407,Z 1183.4,A -85,B 0,C 180,E1 26673.967,E2 26673.967} C_VEL
LIN {X 0,Y 230.589,Z 1132.021,A -85,B 0,C 180,E1 26686.284,E2 26686.284} C_VEL
LIN {X 0,Y 234.151,Z 1124.342,A -85,B 0,C 180,E1 26687.907,E2 26687.907} C_VEL
LIN {X 0,Y 217.911,Z 1162.68,A -85,B 0,C 180,E1 26695.428,E2 26695.428} C_VEL
LIN {X 0,Y 201.935,Z 1190.094,A -85,B 0,C 180,E1 26706.652,E2 26706.652} C_VEL
LIN {X 0,Y 200.906,Z 1191.729,A -85,B 0,C 180,E1 26707.684,E2 26707.684} C_VEL
LIN {X 0,Y 186.359,Z 1202.777,A -85,B 0,C 180,E1 26716.714,E2 26716.714} C_VEL
LIN {X 0,Y 183.931,Z 1205.818,A -85,B 0,C 180,E1 26732.247,E2 26732.247} C_VEL
LIN {X 0,Y 189.898,Z 1195.286,A -85,B 0,C 180,E1 26747.316,E2 26747.316} C_VEL
LIN {X 0,Y 204.178,Z 1170.603,A -85,B 0,C 180,E1 26759.984,E2 26759.984} C_VEL
LIN {X 0,Y 220.734,Z 1134.385,A -85,B 0,C 180,E1 26768.721,E2 26768.721} C_VEL
LIN {X 0,Y 233.423,Z 1088.023,A -85,B 0,C 180,E1 26774.129,E2 26774.129} C_VEL
LIN {X 0,Y 235.838,Z 1058.027,A -85,B 0,C 180,E1 26776.173,E2 26776.173} C_VEL
LIN {X 0,Y 218.937,Z 1014.507,A -85,B 0,C 180,E1 26783.683,E2 26783.683} C_VEL
LIN {X 0,Y 200.751,Z 982.83,A -85,B 0,C 180,E1 26794.567,E2 26794.567} C_VEL
LIN {X 0,Y 189.399,Z 964.85,A -85,B 0,C 180,E1 26806.928,E2 26806.928} C_VEL
LIN {X 0,Y 189.128,Z 970.234,A -85,B 0,C 180,E1 26811.298,E2 26811.298} C_VEL
LIN {X 0,Y 202.125,Z 998.262,A -85,B 0,C 180,E1 26823.725,E2 26823.725} C_VEL
LIN {X 0,Y 218.831,Z 1045.452,A -85,B 0,C 180,E1 26838.146,E2 26838.146} C_VEL
LIN {X 0,Y 234.903,Z 1098.626,A -85,B 0,C 180,E1 26851.239,E2 26851.239} C_VEL
LIN {X 0,Y 235.871,Z 1110.888,A -85,B 0,C 180,E1 26853.726,E2 26853.726} C_VEL
LIN {X 0,Y 206.113,Z 1177.384,A -85,B 0,C 180,E1 26866.166,E2 26866.166} C_VEL
LIN {X 0,Y 187.088,Z 1226.257,A -85,B 0,C 180,E1 26883.02,E2 26883.02} C_VEL
LIN {X 0,Y 181.494,Z 1254.823,A -85,B 0,C 180,E1 26900.495,E2 26900.495} C_VEL
LIN {X 0,Y 180.937,Z 1265.435,A -85,B 0,C 180,E1 26912.522,E2 26912.522} C_VEL
LIN {X 0,Y 183.866,Z 1270.097,A -85,B 0,C 180,E1 26931.924,E2 26931.924} C_VEL
LIN {X 0,Y 219.91,Z 1261.357,A -85,B 0,C 180,E1 26955.862,E2 26955.862} C_VEL
LIN {X 0,Y 183.97,Z 1256.672,A -85,B 0,C 180,E1 26980.78,E2 26980.78} C_VEL
LIN {X 0,Y 179.934,Z 1242.466,A -85,B 0,C 180,E1 27001.256,E2 27001.256} C_VEL
LIN {X 0,Y 185.533,Z 1217.247,A -85,B 0,C 180,E1 27019.961,E2 27019.961} C_VEL
LIN {X 0,Y 202.183,Z 1178.012,A -85,B 0,C 180,E1 27036.293,E2 27036.293} C_VEL
LIN {X 0,Y 223.854,Z 1133.171,A -85,B 0,C 180,E1 27047.342,E2 27047.342} C_VEL
LIN {X 0,Y 208.909,Z 1168.228,A -85,B 0,C 180,E1 27055.621,E2 27055.621} C_VEL
LIN {X 0,Y 192.502,Z 1194.151,A -85,B 0,C 180,E1 27067.893,E2 27067.893} C_VEL
LIN {X 0,Y 186.359,Z 1202.777,A -85,B 0,C 180,E1 27076.714,E2 27076.714} C_VEL
LIN {X 0,Y 175.636,Z 1207.31,A -85,B 0,C 180,E1 27087.342,E2 27087.342} C_VEL
LIN {X 0,Y 180.006,Z 1199.949,A -85,B 0,C 180,E1 27104.524,E2 27104.524} C_VEL
LIN {X 0,Y 193.724,Z 1178.241,A -85,B 0,C 180,E1 27118.541,E2 27118.541} C_VEL
LIN {X 0,Y 211.146,Z 1143.803,A -85,B 0,C 180,E1 27128.499,E2 27128.499} C_VEL
LIN {X 0,Y 225.548,Z 1099.739,A -85,B 0,C 180,E1 27134.634,E2 27134.634} C_VEL
LIN {X 0,Y 230.476,Z 1060.836,A -85,B 0,C 180,E1 27137.493,E2 27137.493} C_VEL
LIN {X 0,Y 214.323,Z 1018.414,A -85,B 0,C 180,E1 27145.251,E2 27145.251} C_VEL
LIN {X 0,Y 197.218,Z 987.802,A -85,B 0,C 180,E1 27156.497,E2 27156.497} C_VEL
LIN {X 0,Y 188.032,Z 973.877,A -85,B 0,C 180,E1 27167.276,E2 27167.276} C_VEL
LIN {X 0,Y 186.982,Z 980.406,A -85,B 0,C 180,E1 27172.96,E2 27172.96} C_VEL
LIN {X 0,Y 200.325,Z 1013.532,A -85,B 0,C 180,E1 27186.483,E2 27186.483} C_VEL
LIN {X 0,Y 216.537,Z 1062.593,A -85,B 0,C 180,E1 27201.011,E2 27201.011} C_VEL
LIN {X 0,Y 229.222,Z 1110.159,A -85,B 0,C 180,E1 27212.657,E2 27212.657} C_VEL
LIN {X 0,Y 199.04,Z 1175.811,A -85,B 0,C 180,E1 27225.165,E2 27225.165} C_VEL
LIN {X 0,Y 181.536,Z 1219.289,A -85,B 0,C 180,E1 27239.345,E2 27239.345} C_VEL
LIN {X 0,Y 173.625,Z 1252.823,A -85,B 0,C 180,E1 27260.06,E2 27260.06} C_VEL
LIN {X 0,Y 173.089,Z 1263.859,A -85,B 0,C 180,E1 27272.636,E2 27272.636} C_VEL
LIN {X 0,Y 176.396,Z 1269.167,A -85,B 0,C 180,E1 27292.904,E2 27292.904} C_VEL
LIN {X 0,Y 209.872,Z 1262.717,A -85,B 0,C 180,E1 27315.992,E2 27315.992} C_VEL
LIN {X 0,Y 174.985,Z 1255.493,A -85,B 0,C 180,E1 27342.378,E2 27342.378} C_VEL
LIN {X 0,Y 172.182,Z 1239.267,A -85,B 0,C 180,E1 27363.84,E2 27363.84} C_VEL
LIN {X 0,Y 179.332,Z 1211.703,A -85,B 0,C 180,E1 27383.096,E2 27383.096} C_VEL
LIN {X 0,Y 198.116,Z 1170.445,A -85,B 0,C 180,E1 27399.257,E2 27399.257} C_VEL
LIN {X 0,Y 213.453,Z 1141.762,A -85,B 0,C 180,E1 27406.848,E2 27406.848} C_VEL
LIN {X 0,Y 215.6,Z 1143.116,A -85,B 0,C 180,E1 27407.91,E2 27407.91} C_VEL
LIN {X 0,Y 197.155,Z 1177.888,A -85,B 0,C 180,E1 27417.56,E2 27417.56} C_VEL
LIN {X 0,Y 182.285,Z 1199.078,A -85,B 0,C 180,E1 27430.428,E2 27430.428} C_VEL
LIN {X 0,Y 176.321,Z 1206.598,A -85,B 0,C 180,E1 27442.461,E2 27442.461} C_VEL
LIN {X 0,Y 175.636,Z 1207.31,A -85,B 0,C 180,E1 27447.342,E2 27447.342} C_VEL
LIN {X 0,Y 169.165,Z 1205.305,A -85,B 0,C 180,E1 27458.94,E2 27458.94} C_VEL
LIN {X 0,Y 180.428,Z 1189.005,A -85,B 0,C 180,E1 27474.733,E2 27474.733} C_VEL
LIN {X 0,Y 198.281,Z 1158.654,A -85,B 0,C 180,E1 27486.715,E2 27486.715} C_VEL
LIN {X 0,Y 215.441,Z 1117.311,A -85,B 0,C 180,E1 27494.276,E2 27494.276} C_VEL
LIN {X 0,Y 225.789,Z 1068.613,A -85,B 0,C 180,E1 27498.309,E2 27498.309} C_VEL
LIN {X 0,Y 213.583,Z 1030.472,A -85,B 0,C 180,E1 27504.833,E2 27504.833} C_VEL
LIN {X 0,Y 197.026,Z 998.043,A -85,B 0,C 180,E1 27515.681,E2 27515.681} C_VEL
LIN {X 0,Y 187.831,Z 983.043,A -85,B 0,C 180,E1 27525.924,E2 27525.924} C_VEL
LIN {X 0,Y 183.394,Z 988.866,A -85,B 0,C 180,E1 27533.531,E2 27533.531} C_VEL
LIN {X 0,Y 196.098,Z 1022.789,A -85,B 0,C 180,E1 27547.182,E2 27547.182} C_VEL
LIN {X 0,Y 211.811,Z 1072.635,A -85,B 0,C 180,E1 27562.056,E2 27562.056} C_VEL
LIN {X 0,Y 221.325,Z 1112.004,A -85,B 0,C 180,E1 27571.907,E2 27571.907} C_VEL
LIN {X 0,Y 183.493,Z 1196.46,A -85,B 0,C 180,E1 27589.524,E2 27589.524} C_VEL
LIN {X 0,Y 170.814,Z 1227.291,A -85,B 0,C 180,E1 27602.961,E2 27602.961} C_VEL
LIN {X 0,Y 165.657,Z 1254.97,A -85,B 0,C 180,E1 27623.556,E2 27623.556} C_VEL
LIN {X 0,Y 164.675,Z 1264.794,A -85,B 0,C 180,E1 27638.076,E2 27638.076} C_VEL
LIN {X 0,Y 178.241,Z 1267.58,A -85,B 0,C 180,E1 27663.739,E2 27663.739} C_VEL
LIN {X 0,Y 200.113,Z 1263.66,A -85,B 0,C 180,E1 27676.03,E2 27676.03} C_VEL
LIN {X 0,Y 166.223,Z 1254.08,A -85,B 0,C 180,E1 27703.88,E2 27703.88} C_VEL
LIN {X 0,Y 164.235,Z 1238.381,A -85,B 0,C 180,E1 27724.026,E2 27724.026} C_VEL
LIN {X 0,Y 171.47,Z 1211.189,A -85,B 0,C 180,E1 27743.528,E2 27743.528} C_VEL
LIN {X 0,Y 190.828,Z 1169.714,A -85,B 0,C 180,E1 27760.207,E2 27760.207} C_VEL
LIN {X 0,Y 201.587,Z 1149.348,A -85,B 0,C 180,E1 27765.727,E2 27765.727} C_VEL
LIN {X 0,Y 207.216,Z 1149.381,A -85,B 0,C 180,E1 27767.541,E2 27767.541} C_VEL
LIN {X 0,Y 187.551,Z 1183.036,A -85,B 0,C 180,E1 27778.14,E2 27778.14} C_VEL
LIN {X 0,Y 173.034,Z 1202.2,A -85,B 0,C 180,E1 27791.997,E2 27791.997} C_VEL
LIN {X 0,Y 167.695,Z 1208.267,A -85,B 0,C 180,E1 27807.304,E2 27807.304} C_VEL
LIN {X 0,Y 169.165,Z 1205.305,A -85,B 0,C 180,E1 27818.94,E2 27818.94} C_VEL
LIN {X 0,Y 168.15,Z 1197.094,A -85,B 0,C 180,E1 27830.697,E2 27830.697} C_VEL
LIN {X 0,Y 185.157,Z 1171.716,A -85,B 0,C 180,E1 27844.395,E2 27844.395} C_VEL
LIN {X 0,Y 203.85,Z 1134.856,A -85,B 0,C 180,E1 27853.365,E2 27853.365} C_VEL
LIN {X 0,Y 217.489,Z 1089.095,A -85,B 0,C 180,E1 27858.688,E2 27858.688} C_VEL
LIN {X 0,Y 219.726,Z 1065.009,A -85,B 0,C 180,E1 27860.555,E2 27860.555} C_VEL
LIN {X 0,Y 205.166,Z 1025.352,A -85,B 0,C 180,E1 27868.868,E2 27868.868} C_VEL
LIN {X 0,Y 190.712,Z 998.15,A -85,B 0,C 180,E1 27880.648,E2 27880.648} C_VEL
LIN {X 0,Y 185.319,Z 991.205,A -85,B 0,C 180,E1 27888.138,E2 27888.138} C_VEL
LIN {X 0,Y 182.325,Z 1003.71,A -85,B 0,C 180,E1 27897.127,E2 27897.127} C_VEL
LIN {X 0,Y 196.43,Z 1046.926,A -85,B 0,C 180,E1 27912.791,E2 27912.791} C_VEL
LIN {X 0,Y 211.475,Z 1099.842,A -85,B 0,C 180,E1 27927.763,E2 27927.763} C_VEL
LIN {X 0,Y 213.437,Z 1113.84,A -85,B 0,C 180,E1 27931.117,E2 27931.117} C_VEL
LIN {X 0,Y 176.198,Z 1197.667,A -85,B 0,C 180,E1 27948.509,E2 27948.509} C_VEL
LIN {X 0,Y 162.824,Z 1227.818,A -85,B 0,C 180,E1 27962.665,E2 27962.665} C_VEL
LIN {X 0,Y 157.784,Z 1255.465,A -85,B 0,C 180,E1 27986,E2 27986} C_VEL
LIN {X 0,Y 156.852,Z 1263.233,A -85,B 0,C 180,E1 27998.481,E2 27998.481} C_VEL
LIN {X 0,Y 171.538,Z 1266.833,A -85,B 0,C 180,E1 28025.248,E2 28025.248} C_VEL
LIN {X 0,Y 189.865,Z 1264.187,A -85,B 0,C 180,E1 28036.27,E2 28036.27} C_VEL
LIN {X 0,Y 158.49,Z 1253.809,A -85,B 0,C 180,E1 28063.07,E2 28063.07} C_VEL
LIN {X 0,Y 156.306,Z 1237.458,A -85,B 0,C 180,E1 28084.231,E2 28084.231} C_VEL
LIN {X 0,Y 164.091,Z 1209.368,A -85,B 0,C 180,E1 28104.654,E2 28104.654} C_VEL
LIN {X 0,Y 184.193,Z 1167.774,A -85,B 0,C 180,E1 28121.573,E2 28121.573} C_VEL
LIN {X 0,Y 190.695,Z 1156.87,A -85,B 0,C 180,E1 28125.005,E2 28125.005} C_VEL
LIN {X 0,Y 198.308,Z 1156.09,A -85,B 0,C 180,E1 28127.324,E2 28127.324} C_VEL
LIN {X 0,Y 178.665,Z 1186.824,A -85,B 0,C 180,E1 28138.272,E2 28138.272} C_VEL
LIN {X 0,Y 163.864,Z 1204.976,A -85,B 0,C 180,E1 28153.736,E2 28153.736} C_VEL
LIN {X 0,Y 160.167,Z 1208.687,A -85,B 0,C 180,E1 28172.581,E2 28172.581} C_VEL
LIN {X 0,Y 168.15,Z 1197.094,A -85,B 0,C 180,E1 28190.697,E2 28190.697} C_VEL
LIN {X 0,Y 172.159,Z 1182.775,A -85,B 0,C 180,E1 28201.551,E2 28201.551} C_VEL
LIN {X 0,Y 192.006,Z 1149.152,A -85,B 0,C 180,E1 28212.429,E2 28212.429} C_VEL
LIN {X 0,Y 208.727,Z 1105.277,A -85,B 0,C 180,E1 28218.985,E2 28218.985} C_VEL
LIN {X 0,Y 214.734,Z 1067.805,A -85,B 0,C 180,E1 28222.066,E2 28222.066} C_VEL
LIN {X 0,Y 201.194,Z 1029.602,A -85,B 0,C 180,E1 28230.587,E2 28230.587} C_VEL
LIN {X 0,Y 187.917,Z 1003.583,A -85,B 0,C 180,E1 28242.723,E2 28242.723} C_VEL
LIN {X 0,Y 184.19,Z 999.82,A -85,B 0,C 180,E1 28248.226,E2 28248.226} C_VEL
LIN {X 0,Y 180.47,Z 1019.29,A -85,B 0,C 180,E1 28260.555,E2 28260.555} C_VEL
LIN {X 0,Y 194.223,Z 1065.253,A -85,B 0,C 180,E1 28276.411,E2 28276.411} C_VEL
LIN {X 0,Y 206.632,Z 1112.22,A -85,B 0,C 180,E1 28289.676,E2 28289.676} C_VEL
LIN {X 0,Y 172.086,Z 1192.407,A -85,B 0,C 180,E1 28305.315,E2 28305.315} C_VEL
LIN {X 0,Y 156.877,Z 1223.893,A -85,B 0,C 180,E1 28319.311,E2 28319.311} C_VEL
LIN {X 0,Y 149.984,Z 1253.452,A -85,B 0,C 180,E1 28345.792,E2 28345.792} C_VEL
LIN {X 0,Y 149.052,Z 1262.655,A -85,B 0,C 180,E1 28361.894,E2 28361.894} C_VEL
LIN {X 0,Y 172.603,Z 1265.387,A -85,B 0,C 180,E1 28391.704,E2 28391.704} C_VEL
LIN {X 0,Y 180.711,Z 1264.495,A -85,B 0,C 180,E1 28395.704,E2 28395.704} C_VEL
LIN {X 0,Y 149.571,Z 1251.485,A -85,B 0,C 180,E1 28425.363,E2 28425.363} C_VEL
LIN {X 0,Y 148.518,Z 1234.859,A -85,B 0,C 180,E1 28445.923,E2 28445.923} C_VEL
LIN {X 0,Y 157.881,Z 1205.031,A -85,B 0,C 180,E1 28467.232,E2 28467.232} C_VEL
LIN {X 0,Y 178.962,Z 1163.597,A -85,B 0,C 180,E1 28483.719,E2 28483.719} C_VEL
LIN {X 0,Y 188.81,Z 1163.33,A -85,B 0,C 180,E1 28487.388,E2 28487.388} C_VEL
LIN {X 0,Y 167.635,Z 1192.979,A -85,B 0,C 180,E1 28499.998,E2 28499.998} C_VEL
LIN {X 0,Y 154.793,Z 1207.415,A -85,B 0,C 180,E1 28515.672,E2 28515.672} C_VEL
LIN {X 0,Y 152.231,Z 1209.645,A -85,B 0,C 180,E1 28532.715,E2 28532.715} C_VEL
LIN {X 0,Y 160.668,Z 1198.172,A -85,B 0,C 180,E1 28551.614,E2 28551.614} C_VEL
LIN {X 0,Y 172.159,Z 1182.775,A -85,B 0,C 180,E1 28561.551,E2 28561.551} C_VEL
LIN {X 0,Y 179.063,Z 1162.997,A -85,B 0,C 180,E1 28570.89,E2 28570.89} C_VEL
LIN {X 0,Y 198.555,Z 1122.043,A -85,B 0,C 180,E1 28578.862,E2 28578.862} C_VEL
LIN {X 0,Y 210.432,Z 1073.664,A -85,B 0,C 180,E1 28583.138,E2 28583.138} C_VEL
LIN {X 0,Y 198.632,Z 1036.843,A -85,B 0,C 180,E1 28591.438,E2 28591.438} C_VEL
LIN {X 0,Y 186.343,Z 1011.15,A -85,B 0,C 180,E1 28603.389,E2 28603.389} C_VEL
LIN {X 0,Y 183.188,Z 1008.151,A -85,B 0,C 180,E1 28608.161,E2 28608.161} C_VEL
LIN {X 0,Y 177.692,Z 1033.662,A -85,B 0,C 180,E1 28623.378,E2 28623.378} C_VEL
LIN {X 0,Y 191.217,Z 1082.09,A -85,B 0,C 180,E1 28639.668,E2 28639.668} C_VEL
LIN {X 0,Y 198.412,Z 1116.042,A -85,B 0,C 180,E1 28649.21,E2 28649.21} C_VEL
LIN {X 0,Y 169.321,Z 1185.263,A -85,B 0,C 180,E1 28661.549,E2 28661.549} C_VEL
LIN {X 0,Y 151.843,Z 1218.797,A -85,B 0,C 180,E1 28675.104,E2 28675.104} C_VEL
LIN {X 0,Y 142.297,Z 1245.408,A -85,B 0,C 180,E1 28699.399,E2 28699.399} C_VEL
LIN {X 0,Y 141.837,Z 1256.782,A -85,B 0,C 180,E1 28713.217,E2 28713.217} C_VEL
LIN {X 0,Y 149.113,Z 1264.818,A -85,B 0,C 180,E1 28740.207,E2 28740.207} C_VEL
LIN {X 0,Y 170.205,Z 1264.355,A -85,B 0,C 180,E1 28755.356,E2 28755.356} C_VEL
LIN {X 0,Y 143.016,Z 1252.662,A -85,B 0,C 180,E1 28781.498,E2 28781.498} C_VEL
LIN {X 0,Y 140.459,Z 1235.192,A -85,B 0,C 180,E1 28804.709,E2 28804.709} C_VEL
LIN {X 0,Y 149.614,Z 1205.447,A -85,B 0,C 180,E1 28827.226,E2 28827.226} C_VEL
LIN {X 0,Y 167.958,Z 1170.171,A -85,B 0,C 180,E1 28842.738,E2 28842.738} C_VEL
LIN {X 0,Y 179.333,Z 1168.83,A -85,B 0,C 180,E1 28846.788,E2 28846.788} C_VEL
LIN {X 0,Y 159.273,Z 1195.593,A -85,B 0,C 180,E1 28859.836,E2 28859.836} C_VEL
LIN {X 0,Y 145.81,Z 1209.529,A -85,B 0,C 180,E1 28877.838,E2 28877.838} C_VEL
LIN {X 0,Y 144.317,Z 1210.601,A -85,B 0,C 180,E1 28892.864,E2 28892.864} C_VEL
LIN {X 0,Y 152.525,Z 1200.179,A -85,B 0,C 180,E1 28911.752,E2 28911.752} C_VEL
LIN {X 0,Y 170.971,Z 1175.737,A -85,B 0,C 180,E1 28926.583,E2 28926.583} C_VEL
LIN {X 0,Y 179.063,Z 1162.997,A -85,B 0,C 180,E1 28930.89,E2 28930.89} C_VEL
LIN {X 0,Y 187.283,Z 1138.036,A -85,B 0,C 180,E1 28938.355,E2 28938.355} C_VEL
LIN {X 0,Y 202.762,Z 1091.793,A -85,B 0,C 180,E1 28943.799,E2 28943.799} C_VEL
LIN {X 0,Y 204.898,Z 1072.278,A -85,B 0,C 180,E1 28945.559,E2 28945.559} C_VEL
LIN {X 0,Y 193.586,Z 1037.892,A -85,B 0,C 180,E1 28954.406,E2 28954.406} C_VEL
LIN {X 0,Y 183.24,Z 1015.401,A -85,B 0,C 180,E1 28966.658,E2 28966.658} C_VEL
LIN {X 0,Y 176.803,Z 1035.06,A -85,B 0,C 180,E1 28979.19,E2 28979.19} C_VEL
LIN {X 0,Y 180.891,Z 1071.97,A -85,B 0,C 180,E1 28994.531,E2 28994.531} C_VEL
LIN {X 0,Y 191.187,Z 1116.542,A -85,B 0,C 180,E1 29008.079,E2 29008.079} C_VEL
LIN {X 0,Y 167.79,Z 1176.463,A -85,B 0,C 180,E1 29017.417,E2 29017.417} C_VEL
LIN {X 0,Y 148.046,Z 1212.486,A -85,B 0,C 180,E1 29030.167,E2 29030.167} C_VEL
LIN {X 0,Y 135.919,Z 1235.564,A -85,B 0,C 180,E1 29048.639,E2 29048.639} C_VEL
LIN {X 0,Y 134.435,Z 1251.633,A -85,B 0,C 180,E1 29068.543,E2 29068.543} C_VEL
LIN {X 0,Y 136.398,Z 1262.005,A -85,B 0,C 180,E1 29093.084,E2 29093.084} C_VEL
LIN {X 0,Y 160.517,Z 1263.745,A -85,B 0,C 180,E1 29115.337,E2 29115.337} C_VEL
LIN {X 0,Y 134.15,Z 1250.113,A -85,B 0,C 180,E1 29143.635,E2 29143.635} C_VEL
LIN {X 0,Y 132.769,Z 1232.298,A -85,B 0,C 180,E1 29166.629,E2 29166.629} C_VEL
LIN {X 0,Y 143.851,Z 1200.728,A -85,B 0,C 180,E1 29190.147,E2 29190.147} C_VEL
LIN {X 0,Y 158.241,Z 1176.266,A -85,B 0,C 180,E1 29202.25,E2 29202.25} C_VEL
LIN {X 0,Y 170.336,Z 1174.523,A -85,B 0,C 180,E1 29206.678,E2 29206.678} C_VEL
LIN {X 0,Y 149.415,Z 1199.676,A -85,B 0,C 180,E1 29220.997,E2 29220.997} C_VEL
LIN {X 0,Y 137.09,Z 1211.313,A -85,B 0,C 180,E1 29240.285,E2 29240.285} C_VEL
LIN {X 0,Y 137.386,Z 1209.876,A -85,B 0,C 180,E1 29259.377,E2 29259.377} C_VEL
LIN {X 0,Y 150.611,Z 1194.85,A -85,B 0,C 180,E1 29278.427,E2 29278.427} C_VEL
LIN {X 0,Y 172.058,Z 1165.719,A -85,B 0,C 180,E1 29292.084,E2 29292.084} C_VEL
LIN {X 0,Y 187.283,Z 1138.036,A -85,B 0,C 180,E1 29298.355,E2 29298.355} C_VEL
LIN {X 0,Y 193.765,Z 1109.173,A -85,B 0,C 180,E1 29304.232,E2 29304.232} C_VEL
LIN {X 0,Y 200.428,Z 1075.409,A -85,B 0,C 180,E1 29307.263,E2 29307.263} C_VEL
LIN {X 0,Y 190.33,Z 1042.763,A -85,B 0,C 180,E1 29316.203,E2 29316.203} C_VEL
LIN {X 0,Y 181.903,Z 1023.888,A -85,B 0,C 180,E1 29327.066,E2 29327.066} C_VEL
LIN {X 0,Y 175.228,Z 1049.987,A -85,B 0,C 180,E1 29341.842,E2 29341.842} C_VEL
LIN {X 0,Y 182.169,Z 1105.46,A -85,B 0,C 180,E1 29362.776,E2 29362.776} C_VEL
LIN {X 0,Y 183.565,Z 1121.112,A -85,B 0,C 180,E1 29366.977,E2 29366.977} C_VEL
LIN {X 0,Y 166.313,Z 1168.174,A -85,B 0,C 180,E1 29373.458,E2 29373.458} C_VEL
LIN {X 0,Y 145.078,Z 1206.105,A -85,B 0,C 180,E1 29385.303,E2 29385.303} C_VEL
LIN {X 0,Y 129.341,Z 1232.069,A -85,B 0,C 180,E1 29404.218,E2 29404.218} C_VEL
LIN {X 0,Y 126.704,Z 1248.142,A -85,B 0,C 180,E1 29426.737,E2 29426.737} C_VEL
LIN {X 0,Y 126.683,Z 1258.441,A -85,B 0,C 180,E1 29447.6,E2 29447.6} C_VEL
LIN {X 0,Y 150.617,Z 1262.772,A -85,B 0,C 180,E1 29475.152,E2 29475.152} C_VEL
LIN {X 0,Y 127.9,Z 1251.21,A -85,B 0,C 180,E1 29499.216,E2 29499.216} C_VEL
LIN {X 0,Y 124.676,Z 1232.465,A -85,B 0,C 180,E1 29525.307,E2 29525.307} C_VEL
LIN {X 0,Y 135.524,Z 1200.93,A -85,B 0,C 180,E1 29550.336,E2 29550.336} C_VEL
LIN {X 0,Y 146.335,Z 1181.821,A -85,B 0,C 180,E1 29560.292,E2 29560.292} C_VEL
LIN {X 0,Y 160.775,Z 1181.086,A -85,B 0,C 180,E1 29567.326,E2 29567.326} C_VEL
LIN {X 0,Y 139.597,Z 1203.367,A -85,B 0,C 180,E1 29582.315,E2 29582.315} C_VEL
LIN {X 0,Y 129.255,Z 1212.258,A -85,B 0,C 180,E1 29599.69,E2 29599.69} C_VEL
LIN {X 0,Y 129.577,Z 1210.838,A -85,B 0,C 180,E1 29619.948,E2 29619.948} C_VEL
LIN {X 0,Y 143.678,Z 1195.838,A -85,B 0,C 180,E1 29639.934,E2 29639.934} C_VEL
LIN {X 0,Y 166.265,Z 1166.734,A -85,B 0,C 180,E1 29653.914,E2 29653.914} C_VEL
LIN {X 0,Y 187.547,Z 1126.672,A -85,B 0,C 180,E1 29662.159,E2 29662.159} C_VEL
LIN {X 0,Y 193.765,Z 1109.173,A -85,B 0,C 180,E1 29664.232,E2 29664.232} C_VEL
LIN {X 0,Y 196.48,Z 1081.555,A -85,B 0,C 180,E1 29668.389,E2 29668.389} C_VEL
LIN {X 0,Y 196.016,Z 1077.944,A -85,B 0,C 180,E1 29669.166,E2 29669.166} C_VEL
LIN {X 0,Y 187.088,Z 1047.163,A -85,B 0,C 180,E1 29678.257,E2 29678.257} C_VEL
LIN {X 0,Y 180.586,Z 1032.718,A -85,B 0,C 180,E1 29687.395,E2 29687.395} C_VEL
LIN {X 0,Y 173.913,Z 1064.906,A -85,B 0,C 180,E1 29704.13,E2 29704.13} C_VEL
LIN {X 0,Y 179.471,Z 1118.407,A -85,B 0,C 180,E1 29723.962,E2 29723.962} C_VEL
LIN {X 0,Y 163.389,Z 1164.26,A -85,B 0,C 180,E1 29730.477,E2 29730.477} C_VEL
LIN {X 0,Y 140.338,Z 1203.538,A -85,B 0,C 180,E1 29742.215,E2 29742.215} C_VEL
LIN {X 0,Y 122.668,Z 1229.894,A -85,B 0,C 180,E1 29761.116,E2 29761.116} C_VEL
LIN {X 0,Y 118.982,Z 1245.718,A -85,B 0,C 180,E1 29786.525,E2 29786.525} C_VEL
LIN {X 0,Y 118.749,Z 1255.898,A -85,B 0,C 180,E1 29806.79,E2 29806.79} C_VEL
LIN {X 0,Y 141.712,Z 1261.367,A -85,B 0,C 180,E1 29835.962,E2 29835.962} C_VEL
LIN {X 0,Y 116.641,Z 1242.514,A -85,B 0,C 180,E1 29870.713,E2 29870.713} C_VEL
LIN {X 0,Y 119.043,Z 1221.189,A -85,B 0,C 180,E1 29895.408,E2 29895.408} C_VEL
LIN {X 0,Y 135.981,Z 1187.039,A -85,B 0,C 180,E1 29918.973,E2 29918.973} C_VEL
LIN {X 0,Y 151.342,Z 1186.17,A -85,B 0,C 180,E1 29927.272,E2 29927.272} C_VEL
LIN {X 0,Y 129.808,Z 1206.688,A -85,B 0,C 180,E1 29943.819,E2 29943.819} C_VEL
LIN {X 0,Y 120.179,Z 1213.968,A -85,B 0,C 180,E1 29966.202,E2 29966.202} C_VEL
LIN {X 0,Y 126.995,Z 1206.771,A -85,B 0,C 180,E1 29990.823,E2 29990.823} C_VEL
LIN {X 0,Y 147.601,Z 1184.988,A -85,B 0,C 180,E1 30009.027,E2 30009.027} C_VEL
LIN {X 0,Y 171.261,Z 1151.048,A -85,B 0,C 180,E1 30020.128,E2 30020.128} C_VEL
LIN {X 0,Y 190.478,Z 1106.41,A -85,B 0,C 180,E1 30026.556,E2 30026.556} C_VEL
LIN {X 0,Y 196.016,Z 1077.944,A -85,B 0,C 180,E1 30029.166,E2 30029.166} C_VEL
LIN {X 0,Y 186.362,Z 1058.244,A -85,B 0,C 180,E1 30037.667,E2 30037.667} C_VEL
LIN {X 0,Y 179.736,Z 1041.113,A -85,B 0,C 180,E1 30047.079,E2 30047.079} C_VEL
LIN {X 0,Y 172.685,Z 1077.729,A -85,B 0,C 180,E1 30065.467,E2 30065.467} C_VEL
LIN {X 0,Y 174.987,Z 1124.739,A -85,B 0,C 180,E1 30082.778,E2 30082.778} C_VEL
LIN {X 0,Y 155.474,Z 1170.35,A -85,B 0,C 180,E1 30089.327,E2 30089.327} C_VEL
LIN {X 0,Y 131.647,Z 1206.837,A -85,B 0,C 180,E1 30101.729,E2 30101.729} C_VEL
LIN {X 0,Y 113.817,Z 1231.384,A -85,B 0,C 180,E1 30122.401,E2 30122.401} C_VEL
LIN {X 0,Y 111.312,Z 1244.626,A -85,B 0,C 180,E1 30148.24,E2 30148.24} C_VEL
LIN {X 0,Y 113.073,Z 1255.588,A -85,B 0,C 180,E1 30173.945,E2 30173.945} C_VEL
LIN {X 0,Y 131.868,Z 1259.542,A -85,B 0,C 180,E1 30196.411,E2 30196.411} C_VEL
LIN {X 0,Y 108.541,Z 1238.52,A -85,B 0,C 180,E1 30234.059,E2 30234.059} C_VEL
LIN {X 0,Y 113.099,Z 1214.475,A -85,B 0,C 180,E1 30260.707,E2 30260.707} C_VEL
LIN {X 0,Y 125.091,Z 1192.085,A -85,B 0,C 180,E1 30277.129,E2 30277.129} C_VEL
LIN {X 0,Y 141.713,Z 1191.004,A -85,B 0,C 180,E1 30287.232,E2 30287.232} C_VEL
LIN {X 0,Y 121.323,Z 1208.721,A -85,B 0,C 180,E1 30303.845,E2 30303.845} C_VEL
LIN {X 0,Y 112.257,Z 1214.919,A -85,B 0,C 180,E1 30325.933,E2 30325.933} C_VEL
LIN {X 0,Y 119.6,Z 1207.747,A -85,B 0,C 180,E1 30352.176,E2 30352.176} C_VEL
LIN {X 0,Y 141.106,Z 1186.468,A -85,B 0,C 180,E1 30370.792,E2 30370.792} C_VEL
LIN {X 0,Y 166.285,Z 1152.085,A -85,B 0,C 180,E1 30382.226,E2 30382.226} C_VEL
LIN {X 0,Y 186.231,Z 1107.53,A -85,B 0,C 180,E1 30388.589,E2 30388.589} C_VEL
LIN {X 0,Y 191.729,Z 1080.505,A -85,B 0,C 180,E1 30391.179,E2 30391.179} C_VEL
LIN {X 0,Y 186.362,Z 1058.244,A -85,B 0,C 180,E1 30397.667,E2 30397.667} C_VEL
LIN {X 0,Y 180.017,Z 1052.47,A -85,B 0,C 180,E1 30404.683,E2 30404.683} C_VEL
LIN {X 0,Y 178.163,Z 1050.797,A -85,B 0,C 180,E1 30407.654,E2 30407.654} C_VEL
LIN {X 0,Y 170.791,Z 1089.777,A -85,B 0,C 180,E1 30426.168,E2 30426.168} C_VEL
LIN {X 0,Y 170.038,Z 1129.44,A -85,B 0,C 180,E1 30440.816,E2 30440.816} C_VEL
LIN {X 0,Y 148.73,Z 1174.098,A -85,B 0,C 180,E1 30447.703,E2 30447.703} C_VEL
LIN {X 0,Y 123.222,Z 1209.577,A -85,B 0,C 180,E1 30461.042,E2 30461.042} C_VEL
LIN {X 0,Y 104.9,Z 1232.962,A -85,B 0,C 180,E1 30484.51,E2 30484.51} C_VEL
LIN {X 0,Y 103.685,Z 1243.443,A -85,B 0,C 180,E1 30510.207,E2 30510.207} C_VEL
LIN {X 0,Y 107.97,Z 1254.541,A -85,B 0,C 180,E1 30539.69,E2 30539.69} C_VEL
LIN {X 0,Y 122.745,Z 1257.586,A -85,B 0,C 180,E1 30556.243,E2 30556.243} C_VEL
LIN {X 0,Y 100.703,Z 1236.568,A -85,B 0,C 180,E1 30594.257,E2 30594.257} C_VEL
LIN {X 0,Y 106.21,Z 1211.064,A -85,B 0,C 180,E1 30623.228,E2 30623.228} C_VEL
LIN {X 0,Y 113.744,Z 1197.014,A -85,B 0,C 180,E1 30634.641,E2 30634.641} C_VEL
LIN {X 0,Y 132.155,Z 1195.395,A -85,B 0,C 180,E1 30647.111,E2 30647.111} C_VEL
LIN {X 0,Y 111.529,Z 1211.519,A -85,B 0,C 180,E1 30665.702,E2 30665.702} C_VEL
LIN {X 0,Y 104.763,Z 1215.379,A -85,B 0,C 180,E1 30693.947,E2 30693.947} C_VEL
LIN {X 0,Y 116.578,Z 1205.075,A -85,B 0,C 180,E1 30719.003,E2 30719.003} C_VEL
LIN {X 0,Y 141.219,Z 1180.659,A -85,B 0,C 180,E1 30736.268,E2 30736.268} C_VEL
LIN {X 0,Y 167.195,Z 1143.564,A -85,B 0,C 180,E1 30746.254,E2 30746.254} C_VEL
LIN {X 0,Y 185.556,Z 1097.382,A -85,B 0,C 180,E1 30751.622,E2 30751.622} C_VEL
LIN {X 0,Y 187.63,Z 1082.436,A -85,B 0,C 180,E1 30753.437,E2 30753.437} C_VEL
LIN {X 0,Y 181.11,Z 1055.68,A -85,B 0,C 180,E1 30762.894,E2 30762.894} C_VEL
LIN {X 0,Y 180.017,Z 1052.47,A -85,B 0,C 180,E1 30764.683,E2 30764.683} C_VEL
LIN {X 0,Y 177.378,Z 1056.331,A -85,B 0,C 180,E1 30767.809,E2 30767.809} C_VEL
LIN {X 0,Y 174.634,Z 1066.008,A -85,B 0,C 180,E1 30770.849,E2 30770.849} C_VEL
LIN {X 0,Y 167.733,Z 1105.674,A -85,B 0,C 180,E1 30788.458,E2 30788.458} C_VEL
LIN {X 0,Y 165.893,Z 1132.021,A -85,B 0,C 180,E1 30798.528,E2 30798.528} C_VEL
LIN {X 0,Y 142.705,Z 1176.679,A -85,B 0,C 180,E1 30805.696,E2 30805.696} C_VEL
LIN {X 0,Y 114.918,Z 1211.939,A -85,B 0,C 180,E1 30820.162,E2 30820.162} C_VEL
LIN {X 0,Y 96.727,Z 1233.095,A -85,B 0,C 180,E1 30844.691,E2 30844.691} C_VEL
LIN {X 0,Y 96.009,Z 1242.127,A -85,B 0,C 180,E1 30872.488,E2 30872.488} C_VEL
LIN {X 0,Y 111.063,Z 1255.013,A -85,B 0,C 180,E1 30913.349,E2 30913.349} C_VEL
LIN {X 0,Y 111.907,Z 1254.601,A -85,B 0,C 180,E1 30917.404,E2 30917.404} C_VEL
LIN {X 0,Y 92.948,Z 1232.32,A -85,B 0,C 180,E1 30957.752,E2 30957.752} C_VEL
LIN {X 0,Y 100.597,Z 1204.869,A -85,B 0,C 180,E1 30988.228,E2 30988.228} C_VEL
LIN {X 0,Y 102.456,Z 1201.647,A -85,B 0,C 180,E1 30991.329,E2 30991.329} C_VEL
LIN {X 0,Y 122.659,Z 1199.365,A -85,B 0,C 180,E1 31006.891,E2 31006.891} C_VEL
LIN {X 0,Y 101.804,Z 1213.979,A -85,B 0,C 180,E1 31027.897,E2 31027.897} C_VEL
LIN {X 0,Y 96.841,Z 1216.337,A -85,B 0,C 180,E1 31054.271,E2 31054.271} C_VEL
LIN {X 0,Y 109.711,Z 1206.052,A -85,B 0,C 180,E1 31081.011,E2 31081.011} C_VEL
LIN {X 0,Y 135.852,Z 1181.667,A -85,B 0,C 180,E1 31098.687,E2 31098.687} C_VEL
LIN {X 0,Y 162.935,Z 1144.609,A -85,B 0,C 180,E1 31108.567,E2 31108.567} C_VEL
LIN {X 0,Y 181.992,Z 1098.268,A -85,B 0,C 180,E1 31113.839,E2 31113.839} C_VEL
LIN {X 0,Y 183.832,Z 1085.162,A -85,B 0,C 180,E1 31115.63,E2 31115.63} C_VEL
LIN {X 0,Y 178.458,Z 1059.968,A -85,B 0,C 180,E1 31125.491,E2 31125.491} C_VEL
LIN {X 0,Y 176.829,Z 1060.418,A -85,B 0,C 180,E1 31127.874,E2 31127.874} C_VEL
LIN {X 0,Y 174.634,Z 1066.008,A -85,B 0,C 180,E1 31130.849,E2 31130.849} C_VEL
LIN {X 0,Y 168.526,Z 1092.046,A -85,B 0,C 180,E1 31138.706,E2 31138.706} C_VEL
LIN {X 0,Y 161.543,Z 1135.532,A -85,B 0,C 180,E1 31156.256,E2 31156.256} C_VEL
LIN {X 0,Y 136.331,Z 1179.922,A -85,B 0,C 180,E1 31163.735,E2 31163.735} C_VEL
LIN {X 0,Y 106.876,Z 1213.793,A -85,B 0,C 180,E1 31178.985,E2 31178.985} C_VEL
LIN {X 0,Y 88.547,Z 1233.162,A -85,B 0,C 180,E1 31204.903,E2 31204.903} C_VEL
LIN {X 0,Y 88.287,Z 1240.66,A -85,B 0,C 180,E1 31235.173,E2 31235.173} C_VEL
LIN {X 0,Y 104.121,Z 1252.641,A -85,B 0,C 180,E1 31275.114,E2 31275.114} C_VEL
LIN {X 0,Y 85.173,Z 1231.959,A -85,B 0,C 180,E1 31314.988,E2 31314.988} C_VEL
LIN {X 0,Y 92.888,Z 1205.826,A -85,B 0,C 180,E1 31349.459,E2 31349.459} C_VEL
LIN {X 0,Y 112.342,Z 1203.69,A -85,B 0,C 180,E1 31367.264,E2 31367.264} C_VEL
LIN {X 0,Y 92.187,Z 1216.113,A -85,B 0,C 180,E1 31390.535,E2 31390.535} C_VEL
LIN {X 0,Y 88.939,Z 1217.293,A -85,B 0,C 180,E1 31414.651,E2 31414.651} C_VEL
LIN {X 0,Y 103.01,Z 1207.027,A -85,B 0,C 180,E1 31443.279,E2 31443.279} C_VEL
LIN {X 0,Y 130.755,Z 1182.673,A -85,B 0,C 180,E1 31461.297,E2 31461.297} C_VEL
LIN {X 0,Y 158.948,Z 1145.656,A -85,B 0,C 180,E1 31471.004,E2 31471.004} C_VEL
LIN {X 0,Y 178.359,Z 1100.371,A -85,B 0,C 180,E1 31476.057,E2 31476.057} C_VEL
LIN {X 0,Y 180.293,Z 1088.228,A -85,B 0,C 180,E1 31477.85,E2 31477.85} C_VEL
LIN {X 0,Y 176.738,Z 1067.396,A -85,B 0,C 180,E1 31486.606,E2 31486.606} C_VEL
LIN {X 0,Y 168.526,Z 1092.046,A -85,B 0,C 180,E1 31498.706,E2 31498.706} C_VEL
LIN {X 0,Y 161.517,Z 1119.557,A -85,B 0,C 180,E1 31506.173,E2 31506.173} C_VEL
LIN {X 0,Y 157.295,Z 1139.216,A -85,B 0,C 180,E1 31513.904,E2 31513.904} C_VEL
LIN {X 0,Y 130.087,Z 1182.819,A -85,B 0,C 180,E1 31521.534,E2 31521.534} C_VEL
LIN {X 0,Y 99.34,Z 1215.062,A -85,B 0,C 180,E1 31537.207,E2 31537.207} C_VEL
LIN {X 0,Y 79.795,Z 1234.03,A -85,B 0,C 180,E1 31567.939,E2 31567.939} C_VEL
LIN {X 0,Y 80.664,Z 1238.504,A -85,B 0,C 180,E1 31597.019,E2 31597.019} C_VEL
LIN {X 0,Y 94.919,Z 1249.455,A -85,B 0,C 180,E1 31636.067,E2 31636.067} C_VEL
LIN {X 0,Y 77.4,Z 1226.591,A -85,B 0,C 180,E1 31680.11,E2 31680.11} C_VEL
LIN {X 0,Y 82.26,Z 1209.911,A -85,B 0,C 180,E1 31704.643,E2 31704.643} C_VEL
LIN {X 0,Y 102.528,Z 1206.75,A -85,B 0,C 180,E1 31725.954,E2 31725.954} C_VEL
LIN {X 0,Y 82.824,Z 1217.92,A -85,B 0,C 180,E1 31753.781,E2 31753.781} C_VEL
LIN {X 0,Y 83.112,Z 1216.618,A -85,B 0,C 180,E1 31785.624,E2 31785.624} C_VEL
LIN {X 0,Y 105.031,Z 1201.853,A -85,B 0,C 180,E1 31812.881,E2 31812.881} C_VEL
LIN {X 0,Y 136.075,Z 1172.828,A -85,B 0,C 180,E1 31827.936,E2 31827.936} C_VEL
LIN {X 0,Y 163.115,Z 1132.409,A -85,B 0,C 180,E1 31835.567,E2 31835.567} C_VEL
LIN {X 0,Y 176.976,Z 1092.904,A -85,B 0,C 180,E1 31839.637,E2 31839.637} C_VEL
LIN {X 0,Y 175.138,Z 1076.897,A -85,B 0,C 180,E1 31846.801,E2 31846.801} C_VEL
LIN {X 0,Y 162.409,Z 1115.531,A -85,B 0,C 180,E1 31864.458,E2 31864.458} C_VEL
LIN {X 0,Y 161.517,Z 1119.557,A -85,B 0,C 180,E1 31866.173,E2 31866.173} C_VEL
LIN {X 0,Y 155.704,Z 1137.243,A -85,B 0,C 180,E1 31870.562,E2 31870.562} C_VEL
LIN {X 0,Y 149.86,Z 1148.925,A -85,B 0,C 180,E1 31872.144,E2 31872.144} C_VEL
LIN {X 0,Y 120.827,Z 1189.149,A -85,B 0,C 180,E1 31880.166,E2 31880.166} C_VEL
LIN {X 0,Y 89.598,Z 1218.123,A -85,B 0,C 180,E1 31897.114,E2 31897.114} C_VEL
LIN {X 0,Y 71.256,Z 1234.553,A -85,B 0,C 180,E1 31931.691,E2 31931.691} C_VEL
LIN {X 0,Y 73.148,Z 1237.276,A -85,B 0,C 180,E1 31962.271,E2 31962.271} C_VEL
LIN {X 0,Y 85.58,Z 1246.194,A -85,B 0,C 180,E1 31994.372,E2 31994.372} C_VEL
LIN {X 0,Y 69.796,Z 1227.782,A -85,B 0,C 180,E1 32033.881,E2 32033.881} C_VEL
LIN {X 0,Y 72.026,Z 1213.847,A -85,B 0,C 180,E1 32058.552,E2 32058.552} C_VEL
LIN {X 0,Y 92.74,Z 1210.52,A -85,B 0,C 180,E1 32087.312,E2 32087.312} C_VEL
LIN {X 0,Y 75.234,Z 1218.863,A -85,B 0,C 180,E1 32112.092,E2 32112.092} C_VEL
LIN {X 0,Y 75.51,Z 1217.58,A -85,B 0,C 180,E1 32147.244,E2 32147.244} C_VEL
LIN {X 0,Y 99.21,Z 1202.942,A -85,B 0,C 180,E1 32175.893,E2 32175.893} C_VEL
LIN {X 0,Y 132.048,Z 1173.841,A -85,B 0,C 180,E1 32190.844,E2 32190.844} C_VEL
LIN {X 0,Y 160.005,Z 1133.479,A -85,B 0,C 180,E1 32198.147,E2 32198.147} C_VEL
LIN {X 0,Y 173.835,Z 1096.524,A -85,B 0,C 180,E1 32201.826,E2 32201.826} C_VEL
LIN {X 0,Y 173.058,Z 1086.573,A -85,B 0,C 180,E1 32206.8,E2 32206.8} C_VEL
LIN {X 0,Y 158.706,Z 1123.918,A -85,B 0,C 180,E1 32223.921,E2 32223.921} C_VEL
LIN {X 0,Y 153.37,Z 1142.4,A -85,B 0,C 180,E1 32231.428,E2 32231.428} C_VEL
LIN {X 0,Y 149.86,Z 1148.925,A -85,B 0,C 180,E1 32232.144,E2 32232.144} C_VEL
LIN {X 0,Y 128.181,Z 1176.85,A -85,B 0,C 180,E1 32233.481,E2 32233.481} C_VEL
LIN {X 0,Y 93.188,Z 1210.666,A -85,B 0,C 180,E1 32246.94,E2 32246.94} C_VEL
LIN {X 0,Y 66.895,Z 1230.126,A -85,B 0,C 180,E1 32275.845,E2 32275.845} C_VEL
LIN {X 0,Y 63.221,Z 1235.557,A -85,B 0,C 180,E1 32303.45,E2 32303.45} C_VEL
LIN {X 0,Y 66.493,Z 1236.383,A -85,B 0,C 180,E1 32330.359,E2 32330.359} C_VEL
LIN {X 0,Y 76.397,Z 1242.249,A -85,B 0,C 180,E1 32356.099,E2 32356.099} C_VEL
LIN {X 0,Y 62.016,Z 1219.989,A -85,B 0,C 180,E1 32403.645,E2 32403.645} C_VEL
LIN {X 0,Y 82.487,Z 1213.704,A -85,B 0,C 180,E1 32447.678,E2 32447.678} C_VEL
LIN {X 0,Y 64.888,Z 1220.615,A -85,B 0,C 180,E1 32482.953,E2 32482.953} C_VEL
LIN {X 0,Y 77.64,Z 1213.589,A -85,B 0,C 180,E1 32525.552,E2 32525.552} C_VEL
LIN {X 0,Y 109.891,Z 1192.217,A -85,B 0,C 180,E1 32547.381,E2 32547.381} C_VEL
LIN {X 0,Y 142.178,Z 1158.364,A -85,B 0,C 180,E1 32557.517,E2 32557.517} C_VEL
LIN {X 0,Y 166.486,Z 1114.205,A -85,B 0,C 180,E1 32562.682,E2 32562.682} C_VEL
LIN {X 0,Y 170.896,Z 1100.051,A -85,B 0,C 180,E1 32564.166,E2 32564.166} C_VEL
LIN {X 0,Y 170.355,Z 1096.295,A -85,B 0,C 180,E1 32566.894,E2 32566.894} C_VEL
LIN {X 0,Y 153.958,Z 1133.926,A -85,B 0,C 180,E1 32584.185,E2 32584.185} C_VEL
LIN {X 0,Y 149.729,Z 1145.443,A -85,B 0,C 180,E1 32588.808,E2 32588.808} C_VEL
LIN {X 0,Y 128.181,Z 1176.85,A -85,B 0,C 180,E1 32593.481,E2 32593.481} C_VEL
LIN {X 0,Y 102.085,Z 1199.929,A -85,B 0,C 180,E1 32596.902,E2 32596.902} C_VEL
LIN {X 0,Y 68.017,Z 1224.254,A -85,B 0,C 180,E1 32619.173,E2 32619.173} C_VEL
LIN {X 0,Y 55.153,Z 1234.577,A -85,B 0,C 180,E1 32662.486,E2 32662.486} C_VEL
LIN {X 0,Y 59.351,Z 1233.881,A -85,B 0,C 180,E1 32692.94,E2 32692.94} C_VEL
LIN {X 0,Y 67.665,Z 1238.407,A -85,B 0,C 180,E1 32715.58,E2 32715.58} C_VEL
LIN {X 0,Y 53.985,Z 1221.309,A -85,B 0,C 180,E1 32760.158,E2 32760.158} C_VEL
LIN {X 0,Y 73.252,Z 1216.088,A -85,B 0,C 180,E1 32806.655,E2 32806.655} C_VEL
LIN {X 0,Y 57.028,Z 1221.564,A -85,B 0,C 180,E1 32841.976,E2 32841.976} C_VEL
LIN {X 0,Y 71.328,Z 1214.564,A -85,B 0,C 180,E1 32889.265,E2 32889.265} C_VEL
LIN {X 0,Y 105.836,Z 1193.211,A -85,B 0,C 180,E1 32910.991,E2 32910.991} C_VEL
LIN {X 0,Y 139.337,Z 1159.4,A -85,B 0,C 180,E1 32920.533,E2 32920.533} C_VEL
LIN {X 0,Y 164.301,Z 1115.31,A -85,B 0,C 180,E1 32925.322,E2 32925.322} C_VEL
LIN {X 0,Y 168.006,Z 1104.559,A -85,B 0,C 180,E1 32926.23,E2 32926.23} C_VEL
LIN {X 0,Y 148.579,Z 1143.691,A -85,B 0,C 180,E1 32944.506,E2 32944.506} C_VEL
LIN {X 0,Y 141.923,Z 1155.366,A -85,B 0,C 180,E1 32946.812,E2 32946.812} C_VEL
LIN {X 0,Y 109.296,Z 1193.606,A -85,B 0,C 180,E1 32954.46,E2 32954.46} C_VEL
LIN {X 0,Y 102.085,Z 1199.929,A -85,B 0,C 180,E1 32956.902,E2 32956.902} C_VEL
LIN {X 0,Y 73.373,Z 1217.298,A -85,B 0,C 180,E1 32964.515,E2 32964.515} C_VEL
LIN {X 0,Y 48.413,Z 1231.552,A -85,B 0,C 180,E1 33002.46,E2 33002.46} C_VEL
LIN {X 0,Y 49.116,Z 1234.129,A -85,B 0,C 180,E1 33039.328,E2 33039.328} C_VEL
LIN {X 0,Y 55.076,Z 1232.238,A -85,B 0,C 180,E1 33064.22,E2 33064.22} C_VEL
LIN {X 0,Y 58.406,Z 1233.866,A -85,B 0,C 180,E1 33075.764,E2 33075.764} C_VEL
LIN {X 0,Y 46.747,Z 1224.285,A -85,B 0,C 180,E1 33110.842,E2 33110.842} C_VEL
LIN {X 0,Y 62.077,Z 1218.82,A -85,B 0,C 180,E1 33165.674,E2 33165.674} C_VEL
LIN {X 0,Y 49.168,Z 1222.516,A -85,B 0,C 180,E1 33200.682,E2 33200.682} C_VEL
LIN {X 0,Y 65.379,Z 1215.538,A -85,B 0,C 180,E1 33253.669,E2 33253.669} C_VEL
LIN {X 0,Y 102.232,Z 1194.205,A -85,B 0,C 180,E1 33274.874,E2 33274.874} C_VEL
LIN {X 0,Y 137.055,Z 1160.236,A -85,B 0,C 180,E1 33283.689,E2 33283.689} C_VEL
LIN {X 0,Y 161.756,Z 1117.964,A -85,B 0,C 180,E1 33288.047,E2 33288.047} C_VEL
LIN {X 0,Y 143.279,Z 1151.081,A -85,B 0,C 180,E1 33303.166,E2 33303.166} C_VEL
LIN {X 0,Y 109.301,Z 1190.976,A -85,B 0,C 180,E1 33309.722,E2 33309.722} C_VEL
LIN {X 0,Y 73.373,Z 1217.298,A -85,B 0,C 180,E1 33324.515,E2 33324.515} C_VEL
LIN {X 0,Y 45.852,Z 1228.243,A -85,B 0,C 180,E1 33343.987,E2 33343.987} C_VEL
LIN {X 0,Y 41.259,Z 1233.173,A -85,B 0,C 180,E1 33401.125,E2 33401.125} C_VEL
LIN {X 0,Y 49.991,Z 1229.94,A -85,B 0,C 180,E1 33434.488,E2 33434.488} C_VEL
LIN {X 0,Y 39.972,Z 1223.76,A -85,B 0,C 180,E1 33496.601,E2 33496.601} C_VEL
LIN {X 0,Y 52.513,Z 1221.028,A -85,B 0,C 180,E1 33526.503,E2 33526.503} C_VEL
LIN {X 0,Y 41.68,Z 1223.033,A -85,B 0,C 180,E1 33579.964,E2 33579.964} C_VEL
LIN {X 0,Y 69.38,Z 1212.463,A -85,B 0,C 180,E1 33626.35,E2 33626.35} C_VEL
LIN {X 0,Y 109.355,Z 1187.285,A -85,B 0,C 180,E1 33641.89,E2 33641.89} C_VEL
LIN {X 0,Y 143.225,Z 1150.318,A -85,B 0,C 180,E1 33648.171,E2 33648.171} C_VEL
LIN {X 0,Y 153.79,Z 1132.5,A -85,B 0,C 180,E1 33650.446,E2 33650.446} C_VEL
LIN {X 0,Y 140.069,Z 1154.456,A -85,B 0,C 180,E1 33660.256,E2 33660.256} C_VEL
LIN {X 0,Y 104.546,Z 1193.021,A -85,B 0,C 180,E1 33666.185,E2 33666.185} C_VEL
LIN {X 0,Y 63.779,Z 1219.792,A -85,B 0,C 180,E1 33682.562,E2 33682.562} C_VEL
LIN {X 0,Y 45.852,Z 1228.243,A -85,B 0,C 180,E1 33703.987,E2 33703.987} C_VEL
LIN {X 0,Y 31.764,Z 1232.003,A -85,B 0,C 180,E1 33754.486,E2 33754.486} C_VEL
LIN {X 0,Y 39.85,Z 1230.211,A -85,B 0,C 180,E1 33794.422,E2 33794.422} C_VEL
LIN {X 0,Y 37.471,Z 1223.863,A -85,B 0,C 180,E1 33877.702,E2 33877.702} C_VEL
LIN {X 0,Y 40.916,Z 1223.288,A -85,B 0,C 180,E1 33890.222,E2 33890.222} C_VEL
LIN {X 0,Y 39.447,Z 1222.394,A -85,B 0,C 180,E1 33964.573,E2 33964.573} C_VEL
LIN {X 0,Y 77.491,Z 1207.654,A -85,B 0,C 180,E1 33997.7,E2 33997.7} C_VEL
LIN {X 0,Y 117.928,Z 1178.921,A -85,B 0,C 180,E1 34007.921,E2 34007.921} C_VEL
LIN {X 0,Y 145.029,Z 1146.484,A -85,B 0,C 180,E1 34012.431,E2 34012.431} C_VEL
LIN {X 0,Y 137.287,Z 1157.41,A -85,B 0,C 180,E1 34017.185,E2 34017.185} C_VEL
LIN {X 0,Y 100.228,Z 1194.985,A -85,B 0,C 180,E1 34022.335,E2 34022.335} C_VEL
LIN {X 0,Y 58.158,Z 1220.076,A -85,B 0,C 180,E1 34037.131,E2 34037.131} C_VEL
LIN {X 0,Y 31.095,Z 1231.631,A -85,B 0,C 180,E1 34096.589,E2 34096.589} C_VEL
LIN {X 0,Y 31.764,Z 1232.003,A -85,B 0,C 180,E1 34114.486,E2 34114.486} C_VEL
LIN {X 0,Y 27.335,Z 1230.838,A -85,B 0,C 180,E1 34140.185,E2 34140.185} C_VEL
LIN {X 0,Y 30.675,Z 1230.335,A -85,B 0,C 180,E1 34152.493,E2 34152.493} C_VEL
LIN {X 0,Y 31.545,Z 1224.814,A -85,B 0,C 180,E1 34246.59,E2 34246.59} C_VEL
LIN {X 0,Y 33.228,Z 1223.356,A -85,B 0,C 180,E1 34332.35,E2 34332.35} C_VEL
LIN {X 0,Y 74.846,Z 1208.637,A -85,B 0,C 180,E1 34363.319,E2 34363.319} C_VEL
LIN {X 0,Y 116.528,Z 1179.936,A -85,B 0,C 180,E1 34371.733,E2 34371.733} C_VEL
LIN {X 0,Y 132.516,Z 1163.152,A -85,B 0,C 180,E1 34374.173,E2 34374.173} C_VEL
LIN {X 0,Y 93.367,Z 1198.876,A -85,B 0,C 180,E1 34378.577,E2 34378.577} C_VEL
LIN {X 0,Y 46.687,Z 1222.804,A -85,B 0,C 180,E1 34394.775,E2 34394.775} C_VEL
LIN {X 0,Y 24.112,Z 1231.13,A -85,B 0,C 180,E1 34478.759,E2 34478.759} C_VEL
LIN {X 0,Y 27.335,Z 1230.838,A -85,B 0,C 180,E1 34500.185,E2 34500.185} C_VEL
LIN {X 0,Y 22.231,Z 1229.61,A -85,B 0,C 180,E1 34520.08,E2 34520.08} C_VEL
LIN {X 0,Y 14.603,Z 1228.053,A -85,B 0,C 180,E1 34560.759,E2 34560.759} C_VEL
LIN {X 0,Y 20.211,Z 1226.394,A -85,B 0,C 180,E1 34604.899,E2 34604.899} C_VEL
LIN {X 0,Y 18.703,Z 1225.902,A -85,B 0,C 180,E1 34672.681,E2 34672.681} C_VEL
LIN {X 0,Y 58.413,Z 1215.821,A -85,B 0,C 180,E1 34725.387,E2 34725.387} C_VEL
LIN {X 0,Y 92.32,Z 1198.885,A -85,B 0,C 180,E1 34733.688,E2 34733.688} C_VEL
LIN {X 0,Y 45.286,Z 1221.783,A -85,B 0,C 180,E1 34744.544,E2 34744.544} C_VEL
LIN {X 0,Y 15.634,Z 1229.656,A -85,B 0,C 180,E1 34802.528,E2 34802.528} C_VEL
LIN {X 0,Y 19.38,Z 1230.173,A -85,B 0,C 180,E1 34864.297,E2 34864.297} C_VEL
LIN {X 0,Y 16.195,Z 1228.979,A -85,B 0,C 180,E1 34892.65,E2 34892.65} C_VEL
LIN {X 0,Y 14.603,Z 1228.053,A -85,B 0,C 180,E1 34920.759,E2 34920.759} C_VEL
LIN {X 0,Y 10.254,Z 1227.417,A -85,B 0,C 180,E1 34969.998,E2 34969.998} C_VEL
LIN {X 0,Y 11.992,Z 1226.823,A -85,B 0,C 180,E1 35049.013,E2 35049.013} C_VEL
LIN {X 0,Y 48.857,Z 1219.626,A -85,B 0,C 180,E1 35093.238,E2 35093.238} C_VEL
LIN {X 0,Y 9.173,Z 1228.667,A -85,B 0,C 180,E1 35138.168,E2 35138.168} C_VEL
LIN {X 0,Y 9.793,Z 1229.254,A -85,B 0,C 180,E1 35230.557,E2 35230.557} C_VEL
LIN {X 0,Y 10.302,Z 1227.427,A -85,B 0,C 180,E1 35328.684,E2 35328.684} C_VEL
LIN {X 0,Y 11.992,Z 1226.823,A -85,B 0,C 180,E1 35409.013,E2 35409.013} C_VEL
LIN {X 0,Y 13.426,Z 1228.812,A -85,B 0,C 180,E1 35416.591,E2 35416.591} C_VEL
LIN {X 0,Y 13.426,Z 1305,A -85,B 0,C 180,E1 35416.591,E2 35416.591} C_VEL
LIN {X 0,Y 13.426,Z 1305,A -85,B 0,C 180,E1 35416.591,E2 35416.591}

